(* PLC project ArfBotOS, CODESYS CODESYS V3.5 SP22 Patch 3, author Dale Thomas *)
(* stored: creationDateTime 2026-10-03T14:07:57.8103968, version 1.0.0, modificationDateTime 2026-10-03T14:07:57.6510211, organization Thomas Labs *)
(* https://github.com/dalethomas81/ArfBotOS *)

TYPE ST_CncCmd :
STRUCT
	StartPos: 		SMC_PosInfo;				
	OriConvention: 	SMC_ORI_CONVENTION:=SMC_ORI_CONVENTION.ZYZ;
	Filename: 		STRING:='CNC_FromFile.cnc';
	CoordinateType: DUT_Command_CoordinateType:=DUT_Command_CoordinateType.Variable;
	ArrayIndex: 	INT:=GVL.DEC_START_POS;
	ArrayType: 		DUT_Command_ArrayType:=DUT_Command_ArrayType.StoredPosition;
END_STRUCT
END_TYPE

TYPE DUT_Command :
STRUCT
	CommandType: DUT_CommandType;
	CommandString: STRING(GVL.COMMAND_LEN);
	CommandComment: STRING;
END_STRUCT
END_TYPE

TYPE DUT_Program :
STRUCT
	ProgramName: STRING;
	Commands: ARRAY [GVL.PROG_CMDS_ARR_BEG..GVL.PROG_CMDS_ARR_END] OF DUT_Command;
END_STRUCT
END_TYPE

TYPE DUT_StoredPosition :
STRUCT
	Comment: STRING;
	Position: MC_COORD_REF;
END_STRUCT
END_TYPE

TYPE ST_VisionLocate :
STRUCT
    MaxParts: 		UINT:=1; // max number of parts to locate
    MaxOverlap: 	REAL:=0.0; // max overlap of parts. only needed if MaxParts is greater than zero.
    Score: 			REAL:=0.6; // min score
    ToleranceAngle: REAL:=90.0; // max angle +/- to search
	ResultPosition: UINT:=0; // location to store the results in the vision register array
	TemplateName: 	STRING:='Template.jpg'; // name of the template to search
	ScriptFilename: STRING:='FastTemplateMatching.py'; // name of the script that runs the vision program
END_STRUCT
END_TYPE

TYPE ST_VisionCalibrate :
STRUCT
    CheckerSize: REAL:=25.0; // this value is in user units ex mm
    CheckerXCount: UINT:=6; // count of checker blocks in x coordinate
    CheckerYCount: UINT:=9; // count of checker blocks in y coordinate
END_STRUCT
END_TYPE

TYPE ST_VisionCmd :
STRUCT
    CommandType: DUT_Command_VisionType;
    ImageWidth: UINT:=640; // pixel count in x direction (must be supported by camera)
    ImageHeight: UINT:=400; // pixel coutn in y direction (must be supported by camera)
    Calibrate: ST_VisionCalibrate;
    Locate: ST_VisionLocate;
	Timeout: UDINT:=60; // timeout in seconds
END_STRUCT
END_TYPE

TYPE DUT_VisionRegister EXTENDS DUT_StoredPosition :
STRUCT
	Scaling: REAL;
END_STRUCT
END_TYPE

TYPE DUT_Flags :
STRUCT
	Comment: STRING:='';
	Value: BOOL:=FALSE;
END_STRUCT
END_TYPE

TYPE ST_MoveCmd :
STRUCT
	// common
	MoveType: 					DUT_Command_MoveType:=DUT_Command_MoveType.DirectMove;
	Speed: 						LREAL:=0.0;
	CoordSystem: 				SMC_COORD_SYSTEM:=SMC_COORD_SYSTEM.ACS;
	
	// direct/linear moves
	PositionType: 				DUT_Command_PositionType:=DUT_Command_PositionType.AbsolutePosition;
	CoordinateType: 			DUT_Command_CoordinateType:=DUT_Command_CoordinateType.Literal;
	ArrayIndex: 				UINT:=0;
	ArrayType: 					DUT_Command_ArrayType:=DUT_Command_ArrayType.StoredPosition;
	CoordRef: 					MC_COORD_REF:=(X:=0, Y:=0, Z:=0, A:=0, B:=0, C:=0);
	
	// circular moves
	CircularCoordinateType: 	DUT_Command_CoordinateType:=DUT_Command_CoordinateType.Literal;
	CircularArrayIndex: 		UINT:=0;
	CircularArrayType: 			DUT_Command_ArrayType:=DUT_Command_ArrayType.StoredPosition;
	CircleMode: 				SMC_CIRC_MODE:=SMC_CIRC_MODE.CENTER;
	PathChoice: 				MC_CIRC_PATHCHOICE:=MC_CIRC_PATHCHOICE.CLOCKWISE;
	CoordRef2: 					MC_COORD_REF:=(X:=0, Y:=0, Z:=0, A:=0, B:=0, C:=0);
	
END_STRUCT
END_TYPE

TYPE ST_OutputCmd :
STRUCT
	OutputType: DUT_OutputType;
	OutputTarget: INT;
	OutputValue1: LREAL;
END_STRUCT
END_TYPE

TYPE ST_PauseCmd :
STRUCT
	PauseTime: TIME:=T#1S;
END_STRUCT
END_TYPE

TYPE ST_VarSetCmd :
STRUCT
	ArrayType: DUT_Command_ArrayType;
	ArrayIndex: INT;
	Coordinates: MC_COORD_REF;
	XOperType: DUT_VarSetCmd_OperType;
	YOperType: DUT_VarSetCmd_OperType;
	ZOperType: DUT_VarSetCmd_OperType;
	AOperType: DUT_VarSetCmd_OperType;
	BOperType: DUT_VarSetCmd_OperType;
	COperType: DUT_VarSetCmd_OperType;
END_STRUCT
END_TYPE

TYPE ST_LogicCmdIO :
STRUCT
	Input: ARRAY [GVL.DIG_IN_ARR_BEG..GVL.DIG_IN_ARR_END] OF BOOL;
	Output: ARRAY [GVL.DIG_OUT_ARR_BEG..GVL.DIG_OUT_ARR_END] OF BOOL;
	Pwm: ARRAY [GVL.PWM_OUT_ARR_BEG..GVL.PWM_OUT_ARR_END] OF BYTE;
	Register: ARRAY [GVL.REG_ARR_BEG..GVL.REG_ARR_END] OF UDINT;
	Counter: ARRAY [GVL.REG_ARR_BEG..GVL.REG_ARR_END] OF UDINT;
END_STRUCT
END_TYPE

TYPE ST_LogicCmd :
STRUCT
	IF_Condition : E_LogicIfCondition;
	IF_Condition_Idx: INT;
	IF_Condition_Operator: E_LogicIfConditionOperator;
	IF_Condition_Operator_Value: UDINT;
	THEN_Function: E_LogicFunction;
	THEN_Function_Value: UDINT;
	THEN_Function_Idx: INT;
	ELSE_Function: E_LogicFunction;
	ELSE_Function_Idx: INT;
	ELSE_Function_Value: UDINT;
END_STRUCT
END_TYPE

TYPE ST_Buttons :
STRUCT
	Square: BOOL;
	Triangle: BOOL;
	Circle: BOOL;
	Cross: BOOL;
	Share: BOOL;
	Options: BOOL;
	PS: BOOL;
	Touch: BOOL;
	Mic: BOOL;
END_STRUCT
END_TYPE

TYPE ST_Controller :
STRUCT
	Connected: BOOL;
	Joysticks: ST_Joysticks;
	Buttons: ST_Buttons;
	Dpad: ST_Dpad;
	Triggers: ST_Triggers;
	Trackpads: ST_Trackpads;
	Gyroscope: ST_Gyroscope;
	Accelerometer: ST_Accelerometer;
	Battery: ST_Battery;
END_STRUCT
END_TYPE

TYPE ST_Joystick :
STRUCT
	X: USINT;
	Y: USINT;
	ThreeButton: BOOL;
END_STRUCT
END_TYPE

TYPE ST_Dpad :
STRUCT
	Up: BOOL;
	Down: BOOL;
	Left: BOOL;
	Right: BOOL;
END_STRUCT
END_TYPE

TYPE ST_Trigger :
STRUCT
	One: BOOL;
	Two: USINT;
	TwoButton: BOOL;
END_STRUCT
END_TYPE

TYPE ST_Trackpad :
STRUCT
	ID: USINT;
	Active: BOOL;
	X: UINT;
	Y: UINT;
END_STRUCT
END_TYPE

TYPE ST_Triggers :
STRUCT
	Left: ST_Trigger;
	Right: ST_Trigger;
END_STRUCT
END_TYPE

TYPE ST_Trackpads :
STRUCT
	One: ST_Trackpad;
	Two: ST_Trackpad;
END_STRUCT
END_TYPE

TYPE ST_Joysticks :
STRUCT
	Left: ST_Joystick;
	Right: ST_Joystick;
END_STRUCT
END_TYPE

TYPE ST_Gyroscope :
STRUCT
	Pitch: INT;
	Yaw: INT;
	Roll: INT;
END_STRUCT
END_TYPE

TYPE ST_Accelerometer :
STRUCT
	X: INT;
	Y: INT;
	Z: INT;
END_STRUCT
END_TYPE

TYPE ST_Battery :
STRUCT
	State: USINT;
	Level: USINT;
END_STRUCT
END_TYPE

TYPE DUT_PositionController :
STRUCT
	fKp: LREAL;
	fPartVelPilotControl: LREAL;
	fDeadTime: LREAL;
	fMaxPositionDiff: LREAL;
	fSWMaxVelocity: LREAL;
	fSWMaxAcceleration: LREAL;
	fSWMaxDeceleration: LREAL;
	fSWMaxJerk: LREAL;
END_STRUCT
END_TYPE

TYPE DUT_GroupStatus :
STRUCT
	Valid: BOOL;
	Busy: BOOL;
	Error: BOOL;
	ErrorID: SMC_ERROR;
	GroupMoving: BOOL;
	GroupHoming: BOOL;
	GroupErrorStop: BOOL;
	GroupStandby: BOOL;
	GroupStopping: BOOL;
	GroupDisabled: BOOL;
	TrackingDynamicCS: BOOL;
	InSync: BOOL;
	ActiveMovementId: SMC_Movement_Id;
	FirstReferencedMovementId: SMC_Movement_Id;
	LastAcceptedMovementId: SMC_Movement_Id;
	PositionLag: LREAL;
	OrientationLag: LREAL;
END_STRUCT
END_TYPE

{attribute 'qualified_only'}
{attribute 'strict'}
TYPE E_ControllerPlayerID :
(
	Player1 := 4,
	Player2 := 10,
	Player3 := 21,
	Player4 := 27,
	PlayerAll := 31
);
END_TYPE

{attribute 'qualified_only'}
{attribute 'strict'}
TYPE E_ControllerBrightness :
(
	High := 0,
	Med := 1,
	Low := 2
);
END_TYPE

{attribute 'qualified_only'}
{attribute 'strict'}
TYPE E_ControllerMotor :
(
	Left := 0,
	Right := 1
);
END_TYPE

{attribute 'qualified_only'}
{attribute 'strict'}
TYPE E_ControllerTriggerMode :
(
	Off := 0, // no resistance
	Rigid := 1, // continous resistance
	Pulse := 2, // section resistance
	Rigid_A := 3,
	Rigid_B := 4,
	Rigid_AB := 5,
	Pulse_A := 6,
	Pulse_AB := 7,
	Calibration := 8
);
END_TYPE

{attribute 'qualified_only'}
{attribute 'strict'}
TYPE E_ControllerTrigger :
(
	Left := 0,
	Right := 1
);
END_TYPE

{attribute 'qualified_only'}
{attribute 'strict'}
TYPE E_ControllerTriggerForceParameter :
(
	One := 0,
	Two := 1,
	Three := 2,
	Four := 3,
	Five := 4,
	Six := 5,
	Seven := 6
);
END_TYPE

{attribute 'qualified_only'}
{attribute 'strict'}
TYPE E_Pose :
(
	One := 0,
	Two := 1,
	Three := 2,
	Four := 3,
	Five := 4
);
END_TYPE

TYPE DUT_AxisEnabled :
STRUCT
	J1: BOOL;
	J2: BOOL;
	J3: BOOL;
	J4: BOOL;
	J5: BOOL;
	J6: BOOL;
END_STRUCT
END_TYPE

INTERFACE ITFModule
METHOD M_Start
VAR_INPUT
END_VAR
END_METHOD
METHOD M_Stop
VAR_INPUT
END_VAR
END_METHOD
METHOD M_Home
VAR_INPUT
END_VAR
END_METHOD
METHOD M_Abort
VAR_INPUT
END_VAR
END_METHOD
METHOD M_Hold
VAR_INPUT
END_VAR
END_METHOD
{attribute 'monitoring' := 'variable'}
PROPERTY PropCurrentState : PACK_ML.State
END_PROPERTY
{attribute 'monitoring' := 'variable'}
PROPERTY PropBusy : BOOL
END_PROPERTY
{attribute 'monitoring' := 'variable'}
PROPERTY PropError : BOOL
END_PROPERTY
{attribute 'monitoring' := 'variable'}
PROPERTY PropErrDescription : STRING
END_PROPERTY
END_INTERFACE

TYPE StringByteArray : UNION
  bArray : ARRAY[0..254] OF BYTE;
  sString : STRING(255);
END_UNION;
END_TYPE

PROGRAM _00_Main
VAR
	//
    TaskInfo : POINTER TO CmpIecTask.Task_Info2;
    TaskHandle: CmpIecTask.RTS_IEC_HANDLE;
    Result: CmpIecTask.RTS_IEC_RESULT;
    
	// group handler for all motion fbs
	GroupHandler: FB_GroupHandler;
	
	// tuning
	MoveDistance: LREAL := 5.0;
	MoveRelative: ARRAY[0..5] OF MC_MoveRelative;
	EstimateDeadTime: ARRAY[0..5] OF SMC_EstimateDeadTime;
	TuneStart: ARRAY[0..5] OF BOOL;
	TraceStart: ARRAY[0..5] OF BOOL;
	TraceStop: ARRAY[0..5] OF BOOL;
	SetTuningMoveValues: BOOL:=TRUE;
	fCycleTimeMs: LREAL; (* MainTask / SoftMotion bus cycle, ms *)
	fMeasuredLagMs: ARRAY[0..5] OF LREAL;
	fEstimatedDeadTimeRaw: ARRAY[0..5] OF LREAL; (* unclamped SMC_EstimateDeadTime median *)
	fSuggestedDeadTime: ARRAY[0..5] OF LREAL; (* D in MainTask cycles, clamped to (0, 20] *)
	nDeadTimeSamples: ARRAY[0..5] OF INT;
	bDeadTimeSuggested: ARRAY[0..5] OF BOOL;
	UseSuggestedD: ARRAY[0..5] OF BOOL;
	sDeadTimeHelp: ARRAY[0..5] OF STRING(255);
	fKpPeakLag: ARRAY[0..5] OF LREAL;
	fKpCruiseLag: ARRAY[0..5] OF LREAL;
	fKpFinalLag: ARRAY[0..5] OF LREAL;
	fKpOvershoot: ARRAY[0..5] OF LREAL;
	fKpUndershoot: ARRAY[0..5] OF LREAL;
	nKpReversals: ARRAY[0..5] OF INT;
	nKpVelReversals: ARRAY[0..5] OF INT;
	fSuggestedKp: ARRAY[0..5] OF LREAL;
	bKpSuggested: ARRAY[0..5] OF BOOL;
	UseSuggestedKp: ARRAY[0..5] OF BOOL;
	RaiseKp: ARRAY[0..5] OF BOOL;
	LowerKp: ARRAY[0..5] OF BOOL;
	sKpVerdict: ARRAY[0..5] OF STRING(16);
	sKpHelp: ARRAY[0..5] OF STRING(255);
	
	// homing
	ProcessHome: FB_HomingProcessor;
	HomingStatusText: STRING(255);
	
	// jogging
	ProcessJog: FB_JogProcessor;
	JogStatusText: STRING(255);
	ButtonTextIndex: INT:=0;
	
	// cnc
	VisuStruct3DControl_J: VisuStruct3DControl;
	TrackPosition: FB_PositionTracker;
	
	// program processor
	ProcessPrograms: FB_ProgramProcessor;
	ProcessCommand_ActiveProgram: UINT := 0;
	ActiveCommandDetails: STRING(255):='';
	
	// controller
	Controller: FB_Controller;
	
	//
	EnableRtrig: R_TRIG;
	EnableFtrig: F_TRIG;
	_i, _j, _k: INT;
	BuildTests: BOOL:=FALSE;
	FirstScan: BOOL:=TRUE;

END_VAR

                    
{region "utility"}
    (* Get the current task info *)
    {IF defined (IsSimulationMode)}
        GVL.dwMainInterval := 1000;
    {ELSE}
        TaskHandle := CmpIecTask.IecTaskGetCurrent(ADR(Result));
        TaskInfo := CmpIecTask.IecTaskGetInfo3(TaskHandle, ADR(Result));
        GVL.dwMainInterval := TaskInfo^.dwInterval;
    {END_IF}
    
	GVL.ResetRtrig(CLK:=GVL.Reset);
	IF GVL.ResetRtrig.Q THEN
		GVL.Reset := FALSE;
        AlarmManager.AlarmGlobals.g_AlarmHandler.AcknowledgeAll();
        //AlarmManager.AlarmGlobals.g_AlarmHandler.AcknowledgeAllOfGroup(Alm_AlarmConfiguration_Alarmgroup_IDs.ID_Processors); // only processors
	END_IF
	
	GVL.LicenseStatus();

	IF FirstScan THEN
		M_Init();	
	END_IF
	
	IF BuildTests THEN
		BuildTests := FALSE;
		M_BuildTests();
	END_IF
	
	EnableRtrig(CLK:=GVL.PowerOn);
	EnableFtrig(CLK:=GVL.PowerOn);
	IF EnableRTrig.Q THEN
		GVL.Enable := TRUE;
	END_IF
	IF EnableFTrig.Q THEN
		GVL.Enable := FALSE;
	END_IF
{endregion}
     
{region "methods"}
	_M_GroupHandler();
    _M_Jogging();
    _M_Homing();
    _M_Cnc();
    _M_Processor();
	_M_Controller();
	_M_Tuning();
{endregion}

// do not put anything below this
FirstScan:=FALSE;
                  

METHOD PUBLIC M_Init : BOOL
VAR_INPUT
END_VAR
VAR
    // release
    _hRelease : SysTypes.RTS_IEC_HANDLE;
    _udiReleaseResult : SysTypes.RTS_IEC_RESULT;
    _udiReleaseRead : LWORD;
    _abyRelease : ARRAY[0..80] OF BYTE;
    _iRelease : INT;
    _nRelease : UDINT;
    _pReleaseLen : POINTER TO BYTE;
END_VAR
                          // get release tag to display on HMI
GVL_Version.sRelease := '';
_hRelease := SysFile.SysFileOpen(
    szFile := 'Application/RELEASE',
    am := SysFile.ACCESS_MODE.AM_READ,
    pResult := ADR(_udiReleaseResult));
IF _hRelease <> SysTypes.RTS_INVALID_HANDLE THEN
    _udiReleaseRead := SysFile.SysFileRead(
        hFile := _hRelease,
        pbyBuffer := ADR(_abyRelease),
        ulSize := SIZEOF(_abyRelease) - 1,
        pResult := ADR(_udiReleaseResult));
    SysFile.SysFileClose(_hRelease);

    _nRelease := LWORD_TO_UDINT(_udiReleaseRead);
    IF _nRelease > 80 THEN
        _nRelease := 80;
    END_IF
    WHILE _nRelease > 0 AND
        (_abyRelease[_nRelease - 1] = 10
        OR _abyRelease[_nRelease - 1] = 13
        OR _abyRelease[_nRelease - 1] = 0) DO
        _nRelease := _nRelease - 1;
    END_WHILE

    MemUtils.MemCpy(
        pbyDest := ADR(GVL_Version.sRelease),
        pbySrc := ADR(_abyRelease),
        dwSize := UDINT_TO_DWORD(_nRelease));
    _pReleaseLen := ADR(GVL_Version.sRelease) - 1;
    _pReleaseLen^ := UDINT_TO_BYTE(_nRelease);
    
    GVL_Version.sVersionLine := CONCAT(
        CONCAT('Installer ', GVL_Version.sRelease),
        CONCAT('  PLC ', GVL_Version.sPlcVersion));
    
END_IF
IF GVL_Version.sRelease = '' THEN
    GVL_Version.sVersionLine := 'unknown version';
    
END_IF

// check if arfbot has been initialized
IF NOT PersistentVars.Flags[GVL.INIT_POS_IDX].Value THEN
	// poses
	PersistentVars.Flags[GVL.HOM_TO_POSE_IDX].Value := FALSE;
	PersistentVars.StoredPositions[GVL.POSE_1_IDX].Position.X := 0.0;
	PersistentVars.StoredPositions[GVL.POSE_1_IDX].Position.Y := 0.0;
	PersistentVars.StoredPositions[GVL.POSE_1_IDX].Position.Z := -30.0;
	PersistentVars.StoredPositions[GVL.POSE_1_IDX].Position.A := 0.0;
	PersistentVars.StoredPositions[GVL.POSE_1_IDX].Position.B := -30.0;
	PersistentVars.StoredPositions[GVL.POSE_1_IDX].Position.C := 0.0;
	
	PersistentVars.StoredPositions[GVL.POSE_2_IDX].Position.X := 0.0;
	PersistentVars.StoredPositions[GVL.POSE_2_IDX].Position.Y := 30.0;
	PersistentVars.StoredPositions[GVL.POSE_2_IDX].Position.Z := -30.0;
	PersistentVars.StoredPositions[GVL.POSE_2_IDX].Position.A := 0.0;
	PersistentVars.StoredPositions[GVL.POSE_2_IDX].Position.B := 30.0;
	PersistentVars.StoredPositions[GVL.POSE_2_IDX].Position.C := 0.0;
	
	PersistentVars.StoredPositions[GVL.POSE_3_IDX].Position.X := 0.0;
	PersistentVars.StoredPositions[GVL.POSE_3_IDX].Position.Y := 0.0;
	PersistentVars.StoredPositions[GVL.POSE_3_IDX].Position.Z := 0.0;
	PersistentVars.StoredPositions[GVL.POSE_3_IDX].Position.A := 0.0;
	PersistentVars.StoredPositions[GVL.POSE_3_IDX].Position.B := 90.0;
	PersistentVars.StoredPositions[GVL.POSE_3_IDX].Position.C := 0.0;
	
	PersistentVars.StoredPositions[GVL.POSE_4_IDX].Position.X := 0.0;
	PersistentVars.StoredPositions[GVL.POSE_4_IDX].Position.Y := 0.0;
	PersistentVars.StoredPositions[GVL.POSE_4_IDX].Position.Z := 0.0;
	PersistentVars.StoredPositions[GVL.POSE_4_IDX].Position.A := 0.0;
	PersistentVars.StoredPositions[GVL.POSE_4_IDX].Position.B := 0.0;
	PersistentVars.StoredPositions[GVL.POSE_4_IDX].Position.C := 0.0;
	
	PersistentVars.StoredPositions[GVL.POSE_5_IDX].Position.X := 0.0;
	PersistentVars.StoredPositions[GVL.POSE_5_IDX].Position.Y := 0.0;
	PersistentVars.StoredPositions[GVL.POSE_5_IDX].Position.Z := 0.0;
	PersistentVars.StoredPositions[GVL.POSE_5_IDX].Position.A := 0.0;
	PersistentVars.StoredPositions[GVL.POSE_5_IDX].Position.B := 0.0;
	PersistentVars.StoredPositions[GVL.POSE_5_IDX].Position.C := 0.0;
		 
	// decoder
	PersistentVars.StoredPositions[GVL.DEC_START_POS].Position.X := 300.0; // TODO need to verify all 6 of these
	PersistentVars.StoredPositions[GVL.DEC_START_POS].Position.Y := 0.0;
	PersistentVars.StoredPositions[GVL.DEC_START_POS].Position.Z := -400.0;
	PersistentVars.StoredPositions[GVL.DEC_START_POS].Position.A := 0.0;
	PersistentVars.StoredPositions[GVL.DEC_START_POS].Position.B := 0.0;
	PersistentVars.StoredPositions[GVL.DEC_START_POS].Position.C := 0.0;
	
	// set homing offsets
	PersistentVars.StoredPositions[GVL.HOM_POS_IDX].Position.X := 179.29; // J1 initial home offset
	PersistentVars.StoredPositions[GVL.HOM_POS_IDX].Position.Y := 36.74; // J2 initial home offset
	PersistentVars.StoredPositions[GVL.HOM_POS_IDX].Position.Z := -59.25; // J3 initial home offset
	PersistentVars.StoredPositions[GVL.HOM_POS_IDX].Position.A := -194.38; // J4 initial home offset
	PersistentVars.StoredPositions[GVL.HOM_POS_IDX].Position.B := -102.41; // J5 initial home offset
	PersistentVars.StoredPositions[GVL.HOM_POS_IDX].Position.C := 166.611; // J6 initial home offset
	
	// set speeds
	PersistentVars.StoredPositions[GVL.SPEEDS_IDX].Position.X := 100.0; // max velocity
	PersistentVars.StoredPositions[GVL.SPEEDS_IDX].Position.Y := 1000.0; // max accel/decel
	PersistentVars.StoredPositions[GVL.SPEEDS_IDX].Position.Z := 1000.0; // max jerk
	PersistentVars.StoredPositions[GVL.SPEEDS_IDX].Position.A := 1.0; // velocity factor
	PersistentVars.StoredPositions[GVL.SPEEDS_IDX].Position.B := 0.05; // accel/decel factor
	PersistentVars.StoredPositions[GVL.SPEEDS_IDX].Position.C := 1.0; // jerk factor
	
	//
	M_BuildTests();
		 
	// indicate initialized
	PersistentVars.Flags[GVL.INIT_POS_IDX].Value := TRUE;
END_IF

//
PersistentVars.StoredPositions[GVL.SPEEDS_IDX].Comment := 'vel, acc, jerk, vel fact, acc fact, jerk fact';
PersistentVars.StoredPositions[GVL.HOM_POS_IDX].Comment := 'Home Offsets J1, J2, J3, J4, J5, J6';
PersistentVars.StoredPositions[GVL.DEC_START_POS].Comment := 'NC Decoder Start Position';
PersistentVars.StoredPositions[GVL.TCP_POS_IDX].Comment := 'TCP Offset';
PersistentVars.StoredPositions[GVL.PC2_POS_IDX].Comment := 'PCS 2 Offset';
PersistentVars.StoredPositions[GVL.PC1_POS_IDX].Comment := 'PCS 1 Offset';
PersistentVars.StoredPositions[GVL.MCS_POS_IDX].Comment := 'MCS Offset';

//	 
PersistentVars.StoredPositions[GVL.POSE_1_IDX].Comment := 'Pose 1 coordinates';
PersistentVars.StoredPositions[GVL.POSE_2_IDX].Comment := 'Pose 2 coordinates';
PersistentVars.StoredPositions[GVL.POSE_3_IDX].Comment := 'Pose 3 coordinates';
PersistentVars.StoredPositions[GVL.POSE_4_IDX].Comment := 'Pose 4 coordinates';
PersistentVars.StoredPositions[GVL.POSE_5_IDX].Comment := 'Pose 5 coordinates';

//
PersistentVars.Flags[GVL.HOM_TO_POSE_IDX].Comment := 'Pose 2 After Home';

PersistentVars.Flags[GVL.INIT_DRV_IDX].Comment := 'Drives Initialized';
PersistentVars.Flags[GVL.INIT_DRV_IDX].Value := FALSE;

//
PersistentVars.Flags[GVL.HOME_COMPLETE].Comment := 'Axes Homed';
PersistentVars.Flags[GVL.HOME_COMPLETE].Value := FALSE;

//
PersistentVars.Flags[GVL.INIT_POS_IDX].Comment := 'Variables Intitialized';
                        
END_METHOD

METHOD PRIVATE _M_Homing : BOOL
VAR_INPUT
END_VAR
                          
ProcessHome(
	J1:= IoConfig_Globals.J1, 
	J2:= IoConfig_Globals.J2, 
	J3:= IoConfig_Globals.J3, 
	J4:= IoConfig_Globals.J4, 
	J5:= IoConfig_Globals.J5, 
	J6:= IoConfig_Globals.J6, 
	AxisGroup:= ArfBotAxisGroup,
	GroupHandler:= GroupHandler, 
	Controller:= Controller, 
	J1_Limit:= _10_Robot.rx_j1_limit, 
	J2_Limit:= _10_Robot.rx_j2_limit, 
	J3_Limit:= _10_Robot.rx_j3_limit, 
	J4_Limit:= _10_Robot.rx_j4_limit, 
	J5_Limit:= _10_Robot.rx_j5_limit, 
	J6_Limit:= _10_Robot.rx_j6_limit, 
	Enable:= GVL.Enable, 
	Reset:= GVL.ResetRtrig.Q, 
	StoredPositions:= PersistentVars.StoredPositions,
	VisionRegisters:= PersistentVars.VisionRegisters,
	Flags:= PersistentVars.Flags,
	Done=> , 
	Busy=> , 
	Error=> , 
	ErrorID=> );

IF ProcessHome.Reset THEN
	HomingStatusText := '';
END_IF
IF ProcessHome.Error THEN
	JogStatusText := CONCAT('Homing Processor Error: ',
						CONCAT(TO_STRING(ProcessHome.ErrorID),
						CONCAT(' ', SMC_ErrorString(ProcessHome.ErrorID,
									SMC_Language_Type.english)))) ;
END_IF
                        
END_METHOD

METHOD PRIVATE _M_Processor : BOOL
VAR_INPUT
END_VAR
                          
IF GVL.ResetRtrig.Q THEN
	ProcessPrograms.M_Home();
END_IF

ProcessPrograms(
	Programs:=PersistentVars.Programs,
	StoredPositions:=PersistentVars.StoredPositions,
	VisionRegisters:=PersistentVars.VisionRegisters,
	Flags:=PersistentVars.Flags,
	J1:=IoConfig_Globals.J1, J2:=IoConfig_Globals.J2, J3:=IoConfig_Globals.J3, J4:=IoConfig_Globals.J4, J5:=IoConfig_Globals.J5, J6:=IoConfig_Globals.J6,
	AxisGroup:= ArfBotAxisGroup,
	GroupHandler:= GroupHandler,
	CmdIO:=GVL.CmdIO,
	Enable:= GVL.Enable AND PersistentVars.Flags[GVL.HOME_COMPLETE].Value AND NOT GVL.xActiveAlarm,
	Error=> ,
	StatusText=>);

IF ProcessPrograms.PropBusy THEN
    // for displaying on the HMI
    // PGM: <number> CMD: <number> Type: <type> Command: <command> Comment: <comment>
    ActiveCommandDetails := CONCAT('PGM: ', UINT_TO_STRING(ProcessPrograms.P_CurrentProgram));
    ActiveCommandDetails := CONCAT(ActiveCommandDetails, ' | CMD: ');
    ActiveCommandDetails := CONCAT(ActiveCommandDetails,
                                    // TODO: the "current" index in this case is actually next
                                    // use a SEL here because I dont want to always do "index minus 1" because this would show a -1 on the HMI when Idle and thats gross
                                    UINT_TO_STRING(SEL(ProcessPrograms.P_CurrentCommandIndex <= 0,
                                                        ProcessPrograms.P_CurrentCommandIndex - 1, // FALSE
                                                        0))); // TRUE
    ActiveCommandDetails := CONCAT(ActiveCommandDetails, ' | ');
    ActiveCommandDetails := CONCAT(ActiveCommandDetails, TO_STRING(ProcessPrograms.P_CurrentCommand.CommandType));
    ActiveCommandDetails := CONCAT(ActiveCommandDetails, ': ');
    ActiveCommandDetails := CONCAT(ActiveCommandDetails, ProcessPrograms.P_CurrentCommand.CommandString);
    IF ProcessPrograms.P_CurrentCommand.CommandType = DUT_CommandType.CncCommand THEN
        ActiveCommandDetails := CONCAT(ActiveCommandDetails, ' | G-Code: ');
        ActiveCommandDetails := CONCAT(ActiveCommandDetails, ProcessPrograms.GCodeLines[0]);
    END_IF
    ActiveCommandDetails := CONCAT(ActiveCommandDetails, ' | Comment: ');
    ActiveCommandDetails := CONCAT(ActiveCommandDetails, ProcessPrograms.P_CurrentCommand.CommandComment);
END_IF

// disable all IO when enable drops
IF EnableFtrig.Q THEN
	FOR _i:=GVL.DIG_OUT_ARR_BEG TO GVL.DIG_OUT_ARR_END BY 1 DO
		GVL.CmdIO.Output[_i] := 0;
	END_FOR
	FOR _i:=GVL.PWM_OUT_ARR_BEG TO GVL.PWM_OUT_ARR_END BY 1 DO
		GVL.CmdIO.Pwm[_i] := 0;
	END_FOR
END_IF
                        
END_METHOD

METHOD PRIVATE _M_Cnc : BOOL
VAR_INPUT
END_VAR
VAR
END_VAR
                          // track position of robot end effector to display on hmi
TrackPosition(
	AxisGroup:=ArfBotAxisGroup,
	J1:=IoConfig_Globals.J1,
	J2:=IoConfig_Globals.J2,
	J3:=IoConfig_Globals.J3,
	J4:=IoConfig_Globals.J4,
	J5:=IoConfig_Globals.J5,
	J6:=IoConfig_Globals.J6,
    OriConvention:= GVL.OriConvention,
	VisuStruct3DTrack=>,
	Arm=>,
	Elbow=>,
	Hand=>);
                        
END_METHOD

METHOD PRIVATE _M_Jogging : BOOL
VAR_INPUT
END_VAR
VAR_STAT
	EnableRtrig: R_TRIG;
	CoordSystemLast: SMC_COORD_SYSTEM;
	ABC_AS_ACSLast: BOOL;
END_VAR
                          
// dont get sleepy
ProcessJog(
	AxisGroup:= ArfBotAxisGroup,
	GroupHandler:= GroupHandler,
	Controller:= Controller,
	Enable:= GVL.Enable,
	Reset:= GVL.ResetRtrig.Q,
	StoredPositions:= PersistentVars.StoredPositions,
	VisionRegisters:= PersistentVars.VisionRegisters,
	Flags:= PersistentVars.Flags,
	ABC_as_ACS=>,
	CoordSystem=>, 
	Enabled=>,
	Position=>, 
	Done=> , 
	Busy=> , 
	Error=> , 
	ErrorID=> );
	
// change the button texts on enable or a change of the coordinate system
EnableRtrig(CLK:=ProcessJog.CoordSystem <> CoordSystemLast
				OR ProcessJog.ABC_as_ACS <> ABC_AS_ACSLast);
IF EnableRtrig.Q THEN
	CoordSystemLast := ProcessJog.CoordSystem;
	ABC_AS_ACSLast := ProcessJog.ABC_as_ACS;
	ButtonTextIndex := F_SetJogButtons(ProcessJog.CoordSystem, ProcessJog.ABC_as_ACS);
END_IF
	
//
IF ProcessJog.Reset THEN
	JogStatusText := '';
END_IF
IF ProcessJog.Error THEN
	JogStatusText := CONCAT('Jog Processor Error: ',
						CONCAT(TO_STRING(ProcessJog.ErrorID),
						CONCAT(' ', SMC_ErrorString(ProcessJog.ErrorID,
									SMC_Language_Type.english)))) ;
END_IF
                        
END_METHOD

METHOD PUBLIC M_BuildTests
VAR_INPUT
END_VAR
VAR
	_i, _j, _k: INT;
END_VAR
                          // taught positions referenced by factory programs
PersistentVars.StoredPositions[40].Position.X := -76.81;
PersistentVars.StoredPositions[40].Position.Y := 1.2;
PersistentVars.StoredPositions[40].Position.Z := -24.93;
PersistentVars.StoredPositions[40].Position.A := -4.74;
PersistentVars.StoredPositions[40].Position.B := 62.93;
PersistentVars.StoredPositions[40].Position.C := 24.21;
PersistentVars.StoredPositions[41].Comment := 'Euler Angle Tool Place Position MCS';
PersistentVars.StoredPositions[41].Position.X := 44.39;
PersistentVars.StoredPositions[41].Position.Y := -285.95;
PersistentVars.StoredPositions[41].Position.Z := 310.15;
PersistentVars.StoredPositions[41].Position.A := 96.6;
PersistentVars.StoredPositions[41].Position.B := 177.75;
PersistentVars.StoredPositions[41].Position.C := -174.21;
PersistentVars.StoredPositions[42].Comment := 'Euler Angle Tool Pick Position MCS';
PersistentVars.StoredPositions[42].Position.X := 43.97;
PersistentVars.StoredPositions[42].Position.Y := -280.38;
PersistentVars.StoredPositions[42].Position.Z := 215.24;
PersistentVars.StoredPositions[42].Position.A := 96.61;
PersistentVars.StoredPositions[42].Position.B := 177.75;
PersistentVars.StoredPositions[42].Position.C := -174.22;

//
FOR _i := GVL.PROG_CMDS_ARR_BEG TO GVL.PROG_CMDS_ARR_END BY 1 DO
	PersistentVars.Programs[0].Commands[_i].CommandType := DUT_CommandType.Disabled;
	PersistentVars.Programs[0].Commands[_i].CommandString := '';
	PersistentVars.Programs[0].Commands[_i].CommandComment := '';
END_FOR
PersistentVars.Programs[0].ProgramName := 'Pick and Place Euler Angle Tool';
PersistentVars.Programs[0].Commands[0].CommandType := DUT_CommandType.MoveCommand;
PersistentVars.Programs[0].Commands[0].CommandString := 'DIR ABS 50.0 ACS VAR STO 35 ';
PersistentVars.Programs[0].Commands[0].CommandComment := 'take on a pose';
PersistentVars.Programs[0].Commands[1].CommandType := DUT_CommandType.VarSetCommand;
PersistentVars.Programs[0].Commands[1].CommandString := 'STO 46 E 0.0 E 0.0 E 0.0 E 0.0 E 0.0 E 0.0 ';
PersistentVars.Programs[0].Commands[1].CommandComment := 'Rotate TCP according to ZYZ convention';
PersistentVars.Programs[0].Commands[3].CommandType := DUT_CommandType.LogicCommand;
PersistentVars.Programs[0].Commands[3].CommandString := 'IF REGISTER 40 EQU 0 THEN JUMP 5 ELSE JUMP 12 ';
PersistentVars.Programs[0].Commands[3].CommandComment := 'determine if pick or place';
PersistentVars.Programs[0].Commands[5].CommandType := DUT_CommandType.MoveCommand;
PersistentVars.Programs[0].Commands[5].CommandString := 'DIR ABS 50.0 MCS VAR STO 42 ';
PersistentVars.Programs[0].Commands[5].CommandComment := 'go to euler angle tool down position';
PersistentVars.Programs[0].Commands[6].CommandType := DUT_CommandType.OutputCommand;
PersistentVars.Programs[0].Commands[6].CommandString := 'DIG 0 1.0 ';
PersistentVars.Programs[0].Commands[6].CommandComment := 'open gripper';
PersistentVars.Programs[0].Commands[7].CommandType := DUT_CommandType.MoveCommand;
PersistentVars.Programs[0].Commands[7].CommandString := 'LIN REL 20.0 TCS LIT 0.0 0.0 25.0 0.0 0.0 0.0 ';
PersistentVars.Programs[0].Commands[7].CommandComment := 'move onto euler angle tool';
PersistentVars.Programs[0].Commands[8].CommandType := DUT_CommandType.OutputCommand;
PersistentVars.Programs[0].Commands[8].CommandString := 'DIG 0 0.0 ';
PersistentVars.Programs[0].Commands[8].CommandComment := 'close gripper';
PersistentVars.Programs[0].Commands[9].CommandType := DUT_CommandType.MoveCommand;
PersistentVars.Programs[0].Commands[9].CommandString := 'LIN REL 20.0 TCS LIT 0.0 0.0 -120.0 0.0 0.0 0.0 ';
PersistentVars.Programs[0].Commands[9].CommandComment := 'pull out tool';
PersistentVars.Programs[0].Commands[10].CommandType := DUT_CommandType.LogicCommand;
PersistentVars.Programs[0].Commands[10].CommandString := 'IF PASS THEN JUMP 16 ';
PersistentVars.Programs[0].Commands[12].CommandType := DUT_CommandType.MoveCommand;
PersistentVars.Programs[0].Commands[12].CommandString := 'DIR ABS 50.0 MCS VAR STO 41 ';
PersistentVars.Programs[0].Commands[12].CommandComment := 'go to euler angle tool up position';
PersistentVars.Programs[0].Commands[13].CommandType := DUT_CommandType.MoveCommand;
PersistentVars.Programs[0].Commands[13].CommandString := 'LIN REL 20.0 TCS LIT 0.0 0.0 120.0 0.0 0.0 0.0 ';
PersistentVars.Programs[0].Commands[13].CommandComment := 'push tool in';
PersistentVars.Programs[0].Commands[14].CommandType := DUT_CommandType.OutputCommand;
PersistentVars.Programs[0].Commands[14].CommandString := 'DIG 0 1.0 ';
PersistentVars.Programs[0].Commands[14].CommandComment := 'open gripper';
PersistentVars.Programs[0].Commands[15].CommandType := DUT_CommandType.MoveCommand;
PersistentVars.Programs[0].Commands[15].CommandString := 'LIN REL 20.0 TCS LIT 0.0 0.0 -25.0 0.0 0.0 0.0 ';
PersistentVars.Programs[0].Commands[15].CommandComment := 'move away from euler angle tool';

//
FOR _i := GVL.PROG_CMDS_ARR_BEG TO GVL.PROG_CMDS_ARR_END BY 1 DO
	PersistentVars.Programs[1].Commands[_i].CommandType := DUT_CommandType.Disabled;
	PersistentVars.Programs[1].Commands[_i].CommandString := '';
	PersistentVars.Programs[1].Commands[_i].CommandComment := '';
END_FOR
PersistentVars.Programs[1].ProgramName := 'Vision Pick and Place';
PersistentVars.Programs[1].Commands[0].CommandType := DUT_CommandType.VarSetCommand;
PersistentVars.Programs[1].Commands[0].CommandString := 'STO 46 E 0.0 E 0.0 E 0.0 E 0.0 E 0.0 E 90.0 ';
PersistentVars.Programs[1].Commands[0].CommandComment := 'Rotate TCP according to ZYZ convention';
PersistentVars.Programs[1].Commands[1].CommandType := DUT_CommandType.MoveCommand;
PersistentVars.Programs[1].Commands[1].CommandString := 'DIR ABS 60.0 ACS VAR STO 40 ';
PersistentVars.Programs[1].Commands[1].CommandComment := 'Take a pose';
PersistentVars.Programs[1].Commands[2].CommandType := DUT_CommandType.VisionCommand;
PersistentVars.Programs[1].Commands[2].CommandString := 'LOC 640 400 15 1 0.0 0.6 180.0 0 Pen.jpg FastTemplateMatching.py ';
PersistentVars.Programs[1].Commands[2].CommandComment := 'Find the object and store the result';
PersistentVars.Programs[1].Commands[3].CommandType := DUT_CommandType.VarSetCommand;
PersistentVars.Programs[1].Commands[3].CommandString := 'VIS 0 M -1.0 M -1.0 E -20.0 M -1.0 N 0.0 N 0.0 ';
PersistentVars.Programs[1].Commands[3].CommandComment := 'Rotate x and y to line up with TCP';
PersistentVars.Programs[1].Commands[4].CommandType := DUT_CommandType.MoveCommand;
PersistentVars.Programs[1].Commands[4].CommandString := 'DIR ABS 50.0 PC1 VAR VIS 0 ';
PersistentVars.Programs[1].Commands[4].CommandComment := 'Move over the object';
PersistentVars.Programs[1].Commands[5].CommandType := DUT_CommandType.OutputCommand;
PersistentVars.Programs[1].Commands[5].CommandString := 'DIG 0 1.0 ';
PersistentVars.Programs[1].Commands[5].CommandComment := 'Open the Gripper';
PersistentVars.Programs[1].Commands[6].CommandType := DUT_CommandType.MoveCommand;
PersistentVars.Programs[1].Commands[6].CommandString := 'LIN REL 50.0 TCS LIT 0.0 0.0 20.0 0.0 0.0 0.0 ';
PersistentVars.Programs[1].Commands[6].CommandComment := 'Move down to the object';
PersistentVars.Programs[1].Commands[7].CommandType := DUT_CommandType.OutputCommand;
PersistentVars.Programs[1].Commands[7].CommandString := 'DIG 0 0.0 ';
PersistentVars.Programs[1].Commands[7].CommandComment := 'Close the Gripper';
PersistentVars.Programs[1].Commands[8].CommandType := DUT_CommandType.PauseCommand;
PersistentVars.Programs[1].Commands[8].CommandString := 'T#1s';
PersistentVars.Programs[1].Commands[8].CommandComment := 'Pause while the gripper closes';
PersistentVars.Programs[1].Commands[9].CommandType := DUT_CommandType.MoveCommand;
PersistentVars.Programs[1].Commands[9].CommandString := 'LIN REL 50.0 TCS LIT 0.0 0.0 -20.0 0.0 0.0 0.0 ';
PersistentVars.Programs[1].Commands[9].CommandComment := 'Pick up the object';
PersistentVars.Programs[1].Commands[10].CommandType := DUT_CommandType.MoveCommand;
PersistentVars.Programs[1].Commands[10].CommandString := 'DIR ABS 50.0 PC1 LIT 0.0 0.0 -50.0 0.0 0.0 90.0 ';
PersistentVars.Programs[1].Commands[10].CommandComment := 'Move to drop position';
PersistentVars.Programs[1].Commands[11].CommandType := DUT_CommandType.OutputCommand;
PersistentVars.Programs[1].Commands[11].CommandString := 'DIG 0 1.0 ';
PersistentVars.Programs[1].Commands[11].CommandComment := 'Open the Gripper';

//
FOR _i := GVL.PROG_CMDS_ARR_BEG TO GVL.PROG_CMDS_ARR_END BY 1 DO
	PersistentVars.Programs[2].Commands[_i].CommandType := DUT_CommandType.Disabled;
	PersistentVars.Programs[2].Commands[_i].CommandString := '';
	PersistentVars.Programs[2].Commands[_i].CommandComment := '';
END_FOR
PersistentVars.Programs[2].ProgramName := 'PCS1 Corners';
PersistentVars.Programs[2].Commands[0].CommandType := DUT_CommandType.VarSetCommand;
PersistentVars.Programs[2].Commands[0].CommandString := 'STO 46 E 0.0 E 0.0 E 0.0 E 180.0 E 180.0 E 0.0 ';
PersistentVars.Programs[2].Commands[0].CommandComment := 'Rotate TCP according to ZYZ convention';
PersistentVars.Programs[2].Commands[1].CommandType := DUT_CommandType.VarSetCommand;
PersistentVars.Programs[2].Commands[1].CommandString := 'STO 48 E 282.23 E -0066.77 E 0195.00 E 0.0 E 0.0 E -0030.00 ';
PersistentVars.Programs[2].Commands[2].CommandType := DUT_CommandType.MoveCommand;
PersistentVars.Programs[2].Commands[2].CommandString := 'DIR ABS 050 PC1 LIT 0 0 0 0 0 0';
PersistentVars.Programs[2].Commands[3].CommandType := DUT_CommandType.MoveCommand;
PersistentVars.Programs[2].Commands[3].CommandString := 'LIN REL 100 TCS LIT 0.0 200.0 0.0 0.0 0.0 0.0';
PersistentVars.Programs[2].Commands[4].CommandType := DUT_CommandType.MoveCommand;
PersistentVars.Programs[2].Commands[4].CommandString := 'LIN REL 100 TCS LIT 00125.00 00000.00 00000.00 00000.00 00000.00 00000.00';
PersistentVars.Programs[2].Commands[5].CommandType := DUT_CommandType.MoveCommand;
PersistentVars.Programs[2].Commands[5].CommandString := 'LIN REL 100 TCS LIT 00000.00 -0200.00 00000.00 00000.00 00000.00 00000.00';
PersistentVars.Programs[2].Commands[6].CommandType := DUT_CommandType.MoveCommand;
PersistentVars.Programs[2].Commands[6].CommandString := 'LIN REL 100 TCS LIT -0125.00 00000.00 00000.00 00000.00 00000.00 00000.00';
PersistentVars.Programs[2].Commands[7].CommandType := DUT_CommandType.MoveCommand;
PersistentVars.Programs[2].Commands[7].CommandString := 'DIR ABS 050 ACS LIT +00 +30 -30 +00 +30 +00';

//
FOR _i := GVL.PROG_CMDS_ARR_BEG TO GVL.PROG_CMDS_ARR_END BY 1 DO
	PersistentVars.Programs[3].Commands[_i].CommandType := DUT_CommandType.Disabled;
	PersistentVars.Programs[3].Commands[_i].CommandString := '';
	PersistentVars.Programs[3].Commands[_i].CommandComment := '';
END_FOR
PersistentVars.Programs[3].ProgramName := 'Cnc Validation';
PersistentVars.Programs[3].Commands[0].CommandType := DUT_CommandType.MoveCommand;
PersistentVars.Programs[3].Commands[0].CommandString := 'DIR ABS 30.0 ACS VAR STO 34 ';
PersistentVars.Programs[3].Commands[1].CommandType := DUT_CommandType.CncCommand;
PersistentVars.Programs[3].Commands[1].CommandString := 'CNC_FromFile.cnc';

//
FOR _i := GVL.PROG_CMDS_ARR_BEG TO GVL.PROG_CMDS_ARR_END BY 1 DO
	PersistentVars.Programs[4].Commands[_i].CommandType := DUT_CommandType.Disabled;
	PersistentVars.Programs[4].Commands[_i].CommandString := '';
	PersistentVars.Programs[4].Commands[_i].CommandComment := '';
END_FOR
PersistentVars.Programs[4].ProgramName := 'Vision Validation';
PersistentVars.Programs[4].Commands[0].CommandType := DUT_CommandType.VisionCommand;
PersistentVars.Programs[4].Commands[0].CommandString := 'LOC 640 400 60 1 0.0 0.8 30.0 10 Template.jpg FastTemplateMatching.py';
PersistentVars.Programs[4].Commands[1].CommandType := DUT_CommandType.VisionCommand;
PersistentVars.Programs[4].Commands[1].CommandString := 'LOC 640 400 60 1 0.0 0.8 30.0 4 strippers2.jpg FastTemplateMatching.py';

//
FOR _i := GVL.PROG_CMDS_ARR_BEG TO GVL.PROG_CMDS_ARR_END BY 1 DO
	PersistentVars.Programs[5].Commands[_i].CommandType := DUT_CommandType.Disabled;
	PersistentVars.Programs[5].Commands[_i].CommandString := '';
	PersistentVars.Programs[5].Commands[_i].CommandComment := '';
END_FOR
PersistentVars.Programs[5].ProgramName := 'VarSet Validation';
PersistentVars.Programs[5].Commands[0].CommandType := DUT_CommandType.VarSetCommand;
PersistentVars.Programs[5].Commands[0].CommandString := 'STO 1 E 6.0 E 5.0 E 4.0 E 3.0 E 2.0 E 1.0 ';
PersistentVars.Programs[5].Commands[1].CommandType := DUT_CommandType.VarSetCommand;
PersistentVars.Programs[5].Commands[1].CommandString := 'VIS 2 1 2 3 4 5 6';
PersistentVars.Programs[5].Commands[2].CommandType := DUT_CommandType.VarSetCommand;
PersistentVars.Programs[5].Commands[2].CommandString := 'FLG 3 1';

//
FOR _i := GVL.PROG_CMDS_ARR_BEG TO GVL.PROG_CMDS_ARR_END BY 1 DO
	PersistentVars.Programs[6].Commands[_i].CommandType := DUT_CommandType.Disabled;
	PersistentVars.Programs[6].Commands[_i].CommandString := '';
	PersistentVars.Programs[6].Commands[_i].CommandComment := '';
END_FOR
PersistentVars.Programs[6].ProgramName := 'Logic Validation';
PersistentVars.Programs[6].Commands[0].CommandType := DUT_CommandType.LogicCommand;
PersistentVars.Programs[6].Commands[0].CommandString := 'IF INPUT 1 EQU 1 THEN OUTPUT 1 1 ELSE OUTPUT 1 0';
PersistentVars.Programs[6].Commands[1].CommandType := DUT_CommandType.LogicCommand;
PersistentVars.Programs[6].Commands[1].CommandString := 'IF INPUT 1 EQU 1 THEN CNTUP 1 ELSE CNTUP 2';
PersistentVars.Programs[6].Commands[2].CommandType := DUT_CommandType.LogicCommand;
PersistentVars.Programs[6].Commands[2].CommandString := 'IF COUNTER 2 GRE 10 THEN NOP ELSE JUMP 0';

//
FOR _i := GVL.PROG_CMDS_ARR_BEG TO GVL.PROG_CMDS_ARR_END BY 1 DO
	PersistentVars.Programs[7].Commands[_i].CommandType := DUT_CommandType.Disabled;
	PersistentVars.Programs[7].Commands[_i].CommandString := '';
	PersistentVars.Programs[7].Commands[_i].CommandComment := '';
END_FOR
PersistentVars.Programs[7].ProgramName := 'Euler Angles Demo';
PersistentVars.Programs[7].Commands[0].CommandType := DUT_CommandType.LogicCommand;
PersistentVars.Programs[7].Commands[0].CommandString := 'IF PASS THEN REGISTER 40 0 ';
PersistentVars.Programs[7].Commands[0].CommandComment := 'Set pick/place register to pick tool';
PersistentVars.Programs[7].Commands[1].CommandType := DUT_CommandType.LogicCommand;
PersistentVars.Programs[7].Commands[1].CommandString := 'IF PASS THEN CALL 0 ';
PersistentVars.Programs[7].Commands[1].CommandComment := 'Call pick and place program';
PersistentVars.Programs[7].Commands[3].CommandType := DUT_CommandType.LogicCommand;
PersistentVars.Programs[7].Commands[3].CommandString := 'IF COUNTER 7 EQU 0 THEN NOP ELSE JUMP 7 ';
PersistentVars.Programs[7].Commands[3].CommandComment := 'apply or jump over';
PersistentVars.Programs[7].Commands[4].CommandType := DUT_CommandType.VarSetCommand;
PersistentVars.Programs[7].Commands[4].CommandString := 'STO 46 E 0.0 E 0.0 E 70.0 E 0.0 E 0.0 E 0.0 ';
PersistentVars.Programs[7].Commands[4].CommandComment := 'offset TCP Z';
PersistentVars.Programs[7].Commands[5].CommandType := DUT_CommandType.LogicCommand;
PersistentVars.Programs[7].Commands[5].CommandString := 'IF PASS THEN JUMP 19 ';
PersistentVars.Programs[7].Commands[5].CommandComment := 'go to move commands';
PersistentVars.Programs[7].Commands[7].CommandType := DUT_CommandType.LogicCommand;
PersistentVars.Programs[7].Commands[7].CommandString := 'IF COUNTER 7 EQU 1 THEN NOP ELSE JUMP 11 ';
PersistentVars.Programs[7].Commands[7].CommandComment := 'apply or jump over';
PersistentVars.Programs[7].Commands[8].CommandType := DUT_CommandType.VarSetCommand;
PersistentVars.Programs[7].Commands[8].CommandString := 'STO 46 E 0.0 E 0.0 E 170.0 E 0.0 E 0.0 E 0.0 ';
PersistentVars.Programs[7].Commands[8].CommandComment := 'offset TCP Z';
PersistentVars.Programs[7].Commands[9].CommandType := DUT_CommandType.LogicCommand;
PersistentVars.Programs[7].Commands[9].CommandString := 'IF PASS THEN JUMP 19 ';
PersistentVars.Programs[7].Commands[9].CommandComment := 'go to move commands';
PersistentVars.Programs[7].Commands[11].CommandType := DUT_CommandType.LogicCommand;
PersistentVars.Programs[7].Commands[11].CommandString := 'IF COUNTER 7 EQU 2 THEN NOP ELSE JUMP 15 ';
PersistentVars.Programs[7].Commands[11].CommandComment := 'apply or jump over';
PersistentVars.Programs[7].Commands[12].CommandType := DUT_CommandType.VarSetCommand;
PersistentVars.Programs[7].Commands[12].CommandString := 'STO 46 E 0.0 E -100.0 E 70.0 E 0.0 E 0.0 E 0.0 ';
PersistentVars.Programs[7].Commands[12].CommandComment := 'offset TCP X and Y';
PersistentVars.Programs[7].Commands[13].CommandType := DUT_CommandType.LogicCommand;
PersistentVars.Programs[7].Commands[13].CommandString := 'IF PASS THEN JUMP 19 ';
PersistentVars.Programs[7].Commands[13].CommandComment := 'go to move commands';
PersistentVars.Programs[7].Commands[15].CommandType := DUT_CommandType.LogicCommand;
PersistentVars.Programs[7].Commands[15].CommandString := 'IF COUNTER 7 EQU 3 THEN NOP ELSE JUMP 29 ';
PersistentVars.Programs[7].Commands[15].CommandComment := 'apply or jump over';
PersistentVars.Programs[7].Commands[16].CommandType := DUT_CommandType.VarSetCommand;
PersistentVars.Programs[7].Commands[16].CommandString := 'STO 46 E 100.0 E 0.0 E 70.0 E 0.0 E 0.0 E 0.0 ';
PersistentVars.Programs[7].Commands[16].CommandComment := 'offset TCP X and Z';
PersistentVars.Programs[7].Commands[17].CommandType := DUT_CommandType.LogicCommand;
PersistentVars.Programs[7].Commands[17].CommandString := 'IF PASS THEN JUMP 19 ';
PersistentVars.Programs[7].Commands[17].CommandComment := 'go to move commands';
PersistentVars.Programs[7].Commands[19].CommandType := DUT_CommandType.MoveCommand;
PersistentVars.Programs[7].Commands[19].CommandString := 'DIR ABS 50.0 ACS VAR STO 35 ';
PersistentVars.Programs[7].Commands[19].CommandComment := 'take on a pose';
PersistentVars.Programs[7].Commands[20].CommandType := DUT_CommandType.MoveCommand;
PersistentVars.Programs[7].Commands[20].CommandString := 'LIN ABS 70.0 TCS LIT 0.0 0.0 0.0 0.0 0.0 -45.0 ';
PersistentVars.Programs[7].Commands[20].CommandComment := 'rotate TCP Z with ZYZ convention';
PersistentVars.Programs[7].Commands[21].CommandType := DUT_CommandType.MoveCommand;
PersistentVars.Programs[7].Commands[21].CommandString := 'LIN ABS 70.0 TCS LIT 0.0 0.0 0.0 0.0 -30.0 0.0 ';
PersistentVars.Programs[7].Commands[21].CommandComment := 'rotate around TCP Y with ZYZ convention';
PersistentVars.Programs[7].Commands[22].CommandType := DUT_CommandType.MoveCommand;
PersistentVars.Programs[7].Commands[22].CommandString := 'LIN ABS 70.0 TCS LIT 0.0 0.0 0.0 90.0 30.0 -90.0 ';
PersistentVars.Programs[7].Commands[22].CommandComment := 'rotate around TCP X with ZYZ convention';
PersistentVars.Programs[7].Commands[23].CommandType := DUT_CommandType.MoveCommand;
PersistentVars.Programs[7].Commands[23].CommandString := 'LIN ABS 70.0 TCS LIT 0.0 0.0 0.0 90.0 -30.0 -90.0 ';
PersistentVars.Programs[7].Commands[23].CommandComment := 'rotate around TCP X with ZYZ convention';
PersistentVars.Programs[7].Commands[24].CommandType := DUT_CommandType.MoveCommand;
PersistentVars.Programs[7].Commands[24].CommandString := 'LIN ABS 70.0 TCS LIT 0.0 0.0 0.0 0.0 30.0 0.0 ';
PersistentVars.Programs[7].Commands[24].CommandComment := 'rotate around TCP Y with ZYZ convention';
PersistentVars.Programs[7].Commands[25].CommandType := DUT_CommandType.MoveCommand;
PersistentVars.Programs[7].Commands[25].CommandString := 'DIR ABS 70.0 ACS VAR STO 35 ';
PersistentVars.Programs[7].Commands[25].CommandComment := 'take on a pose';
PersistentVars.Programs[7].Commands[27].CommandType := DUT_CommandType.LogicCommand;
PersistentVars.Programs[7].Commands[27].CommandString := 'IF PASS THEN CNTUP 7 ';
PersistentVars.Programs[7].Commands[27].CommandComment := 'count up counter';
PersistentVars.Programs[7].Commands[28].CommandType := DUT_CommandType.LogicCommand;
PersistentVars.Programs[7].Commands[28].CommandString := 'IF PASS THEN JUMP 3 ';
PersistentVars.Programs[7].Commands[28].CommandComment := 'go back to start';
PersistentVars.Programs[7].Commands[29].CommandType := DUT_CommandType.LogicCommand;
PersistentVars.Programs[7].Commands[29].CommandString := 'IF PASS THEN CNTRST 7 ';
PersistentVars.Programs[7].Commands[29].CommandComment := 'reset counter back to 0';
PersistentVars.Programs[7].Commands[31].CommandType := DUT_CommandType.LogicCommand;
PersistentVars.Programs[7].Commands[31].CommandString := 'IF PASS THEN REGISTER 40 1 ';
PersistentVars.Programs[7].Commands[31].CommandComment := 'Set pick/place register to place tool';
PersistentVars.Programs[7].Commands[32].CommandType := DUT_CommandType.LogicCommand;
PersistentVars.Programs[7].Commands[32].CommandString := 'IF PASS THEN CALL 0 ';
PersistentVars.Programs[7].Commands[32].CommandComment := 'Call pick and place program';

//
FOR _i := GVL.PROG_CMDS_ARR_BEG TO GVL.PROG_CMDS_ARR_END BY 1 DO
	PersistentVars.Programs[10].Commands[_i].CommandType := DUT_CommandType.Disabled;
	PersistentVars.Programs[10].Commands[_i].CommandString := '';
	PersistentVars.Programs[10].Commands[_i].CommandComment := '';
END_FOR
PersistentVars.Programs[10].ProgramName := 'Pick Glow Stick';
PersistentVars.Programs[10].Commands[0].CommandType := DUT_CommandType.LogicCommand;
PersistentVars.Programs[10].Commands[0].CommandString := 'IF REGISTER 2 EQU 0 THEN NOP ELSE JUMP 5 ';
PersistentVars.Programs[10].Commands[0].CommandComment := 'check if initialized';
PersistentVars.Programs[10].Commands[1].CommandType := DUT_CommandType.VarSetCommand;
PersistentVars.Programs[10].Commands[1].CommandString := 'STO 0 E 0.0 E 0.0 E 0.0 E 0.0 E 0.0 E 0.0 ';
PersistentVars.Programs[10].Commands[1].CommandComment := 'clear out the tcp position';
PersistentVars.Programs[10].Commands[2].CommandType := DUT_CommandType.LogicCommand;
PersistentVars.Programs[10].Commands[2].CommandString := 'IF PASS THEN CNTRST 0 ';
PersistentVars.Programs[10].Commands[2].CommandComment := 'clear column counter';
PersistentVars.Programs[10].Commands[3].CommandType := DUT_CommandType.LogicCommand;
PersistentVars.Programs[10].Commands[3].CommandString := 'IF PASS THEN CNTRST 1 ';
PersistentVars.Programs[10].Commands[3].CommandComment := 'clear row counter';
PersistentVars.Programs[10].Commands[4].CommandType := DUT_CommandType.LogicCommand;
PersistentVars.Programs[10].Commands[4].CommandString := 'IF PASS THEN REGISTER 2 1 ';
PersistentVars.Programs[10].Commands[4].CommandComment := 'mark data initialized';
PersistentVars.Programs[10].Commands[6].CommandType := DUT_CommandType.MoveCommand;
PersistentVars.Programs[10].Commands[6].CommandString := 'DIR ABS 50.0 ACS VAR STO 34 ';
PersistentVars.Programs[10].Commands[6].CommandComment := 'take on a pose';
PersistentVars.Programs[10].Commands[7].CommandType := DUT_CommandType.OutputCommand;
PersistentVars.Programs[10].Commands[7].CommandString := 'DIG 0 1.0 ';
PersistentVars.Programs[10].Commands[7].CommandComment := 'open gripper';
PersistentVars.Programs[10].Commands[8].CommandType := DUT_CommandType.MoveCommand;
PersistentVars.Programs[10].Commands[8].CommandString := 'LIN ABS 50.0 PC1 VAR STO 0 ';
PersistentVars.Programs[10].Commands[8].CommandComment := 'go to the pick position in PCS1';
PersistentVars.Programs[10].Commands[9].CommandType := DUT_CommandType.MoveCommand;
PersistentVars.Programs[10].Commands[9].CommandString := 'LIN REL 50.0 TCS LIT 0.0 0.0 10.0 0.0 0.0 0.0 ';
PersistentVars.Programs[10].Commands[9].CommandComment := 'move into glow stick';
PersistentVars.Programs[10].Commands[10].CommandType := DUT_CommandType.OutputCommand;
PersistentVars.Programs[10].Commands[10].CommandString := 'DIG 0 0.0 ';
PersistentVars.Programs[10].Commands[10].CommandComment := 'close gripper';
PersistentVars.Programs[10].Commands[11].CommandType := DUT_CommandType.MoveCommand;
PersistentVars.Programs[10].Commands[11].CommandString := 'LIN REL 50.0 TCS LIT 160.0 0.0 0.0 0.0 0.0 0.0 ';
PersistentVars.Programs[10].Commands[11].CommandComment := 'pick glow stick out of nest';
PersistentVars.Programs[10].Commands[12].CommandType := DUT_CommandType.MoveCommand;
PersistentVars.Programs[10].Commands[12].CommandString := 'LIN ABS 50.0 PC2 LIT 0.0 0.0 0.0 0.0 0.0 0.0 ';
PersistentVars.Programs[10].Commands[12].CommandComment := 'go to the home position of PCS2';
PersistentVars.Programs[10].Commands[13].CommandType := DUT_CommandType.MoveCommand;
PersistentVars.Programs[10].Commands[13].CommandString := 'LIN REL 50.0 TCS LIT 0.0 0.0 50.0 0.0 0.0 0.0 ';
PersistentVars.Programs[10].Commands[13].CommandComment := 'move into drop position';
PersistentVars.Programs[10].Commands[14].CommandType := DUT_CommandType.OutputCommand;
PersistentVars.Programs[10].Commands[14].CommandString := 'DIG 0 1.0 ';
PersistentVars.Programs[10].Commands[14].CommandComment := 'open gripper';
PersistentVars.Programs[10].Commands[15].CommandType := DUT_CommandType.MoveCommand;
PersistentVars.Programs[10].Commands[15].CommandString := 'LIN ABS 50.0 PC2 LIT 0.0 0.0 0.0 0.0 0.0 0.0 ';
PersistentVars.Programs[10].Commands[15].CommandComment := 'go to the home position of PCS2';
PersistentVars.Programs[10].Commands[17].CommandType := DUT_CommandType.LogicCommand;
PersistentVars.Programs[10].Commands[17].CommandString := 'IF COUNTER 0 LES 3 THEN CNTUP 0 ELSE JUMP 21 ';
PersistentVars.Programs[10].Commands[17].CommandComment := 'increment the column counter';
PersistentVars.Programs[10].Commands[18].CommandType := DUT_CommandType.VarSetCommand;
PersistentVars.Programs[10].Commands[18].CommandString := 'STO 0 N 0.0 A 20.0 N 0.0 N 0.0 N 0.0 N 0.0 ';
PersistentVars.Programs[10].Commands[18].CommandComment := 'add the column width';
PersistentVars.Programs[10].Commands[20].CommandType := DUT_CommandType.LogicCommand;
PersistentVars.Programs[10].Commands[20].CommandString := 'IF PASS THEN JUMP 24 ';
PersistentVars.Programs[10].Commands[20].CommandComment := 'jump over the counter operations';
PersistentVars.Programs[10].Commands[21].CommandType := DUT_CommandType.LogicCommand;
PersistentVars.Programs[10].Commands[21].CommandString := 'IF PASS THEN CNTRST 0 ';
PersistentVars.Programs[10].Commands[21].CommandComment := 'reset the column counter';
PersistentVars.Programs[10].Commands[22].CommandType := DUT_CommandType.LogicCommand;
PersistentVars.Programs[10].Commands[22].CommandString := 'IF PASS THEN CNTUP 1 ';
PersistentVars.Programs[10].Commands[22].CommandComment := 'increment the row counter';
PersistentVars.Programs[10].Commands[23].CommandType := DUT_CommandType.VarSetCommand;
PersistentVars.Programs[10].Commands[23].CommandString := 'STO 0 N 0.0 E 0.0 A 15.0 N 0.0 N 0.0 N 0.0 ';
PersistentVars.Programs[10].Commands[23].CommandComment := 'add the row width. clear column.';

//
FOR _i := GVL.PROG_CMDS_ARR_BEG TO GVL.PROG_CMDS_ARR_END BY 1 DO
	PersistentVars.Programs[15].Commands[_i].CommandType := DUT_CommandType.Disabled;
	PersistentVars.Programs[15].Commands[_i].CommandString := '';
	PersistentVars.Programs[15].Commands[_i].CommandComment := '';
END_FOR
PersistentVars.Programs[15].ProgramName := 'Gimbal 1';
PersistentVars.Programs[15].Commands[0].CommandType := DUT_CommandType.VarSetCommand;
PersistentVars.Programs[15].Commands[0].CommandString := 'STO 43 N 0.0 E 250.0 E 250.0 N 0.0 E 1.0e-2 E 1.0e-1 ';
PersistentVars.Programs[15].Commands[0].CommandComment := 'set velocity, acceleration, and jerk';
PersistentVars.Programs[15].Commands[1].CommandType := DUT_CommandType.VarSetCommand;
PersistentVars.Programs[15].Commands[1].CommandString := 'STO 43 E 100.0 E 1000.0 E 1000.0 E 1.0 E 1.0 E 1.0 ';
PersistentVars.Programs[15].Commands[1].CommandComment := 'set velocity, acceleration, and jerk';
PersistentVars.Programs[15].Commands[3].CommandType := DUT_CommandType.MoveCommand;
PersistentVars.Programs[15].Commands[3].CommandString := 'DIR ABS 30.0 ACS LIT -19.65 30.42 -55.18 0.0 4.04 0.0 ';
PersistentVars.Programs[15].Commands[3].CommandComment := 'Taught position';
PersistentVars.Programs[15].Commands[6].CommandType := DUT_CommandType.VarSetCommand;
PersistentVars.Programs[15].Commands[6].CommandString := 'STO 46 E 0.0 E 0.0 E 300.0 E 0.0 E 0.0 E 0.0 ';
PersistentVars.Programs[15].Commands[6].CommandComment := 'offset the TCP Z';
PersistentVars.Programs[15].Commands[7].CommandType := DUT_CommandType.MoveCommand;
PersistentVars.Programs[15].Commands[7].CommandString := 'LIN ABS 20.0 TCS LIT 0.0 0.0 0.0 0.0 -30.0 0.0 ';
PersistentVars.Programs[15].Commands[7].CommandComment := 'rotate around TCP Y';
PersistentVars.Programs[15].Commands[8].CommandType := DUT_CommandType.MoveCommand;
PersistentVars.Programs[15].Commands[8].CommandString := 'LIN ABS 20.0 TCS LIT 0.0 0.0 0.0 90.0 60.0 -90.0 ';
PersistentVars.Programs[15].Commands[8].CommandComment := 'rotate around TCP X with z$' y z$'$'';
PersistentVars.Programs[15].Commands[10].CommandType := DUT_CommandType.MoveCommand;
PersistentVars.Programs[15].Commands[10].CommandString := 'DIR ABS 30.0 ACS LIT -19.65 30.42 -55.18 0.0 4.04 0.0 ';
PersistentVars.Programs[15].Commands[10].CommandComment := 'Taught position';
PersistentVars.Programs[15].Commands[12].CommandType := DUT_CommandType.VarSetCommand;
PersistentVars.Programs[15].Commands[12].CommandString := 'STO 43 E 100.0 E 1000.0 E 1000.0 E 1.0 E 1.0 E 1.0 ';
PersistentVars.Programs[15].Commands[12].CommandComment := 'set velocity, acceleration, and jerk';
                        
END_METHOD

METHOD PRIVATE _M_Controller : BOOL
VAR_INPUT
END_VAR
VAR_STAT
	_PowerRtrig: R_TRIG;
	_PowerFtrig: F_TRIG;
	_PowerTimerRtrig: R_TRIG;
	_PowerTimer: TON:=(PT:=T#1S);
	_PsButtonRtrig: R_TRIG;
	_PsButtonFtrig: F_TRIG;
	_PsButtonTimer: TON:=(PT:=T#2S);
	_PsButtonTimerRtrig: R_TRIG;
	_Reseting: BOOL;
END_VAR
                          
// dont get sleepy
Controller(sIpAddress:= '127.0.0.1', uPort:= 50013);

// put two fingers on the trackpad for 3 seconds to toggle power
_PowerTimer(IN:=Controller.P_State.Connected
				AND Controller.P_State.Buttons.Touch
				AND Controller.P_State.Trackpads.One.Active 
				AND Controller.P_State.Trackpads.Two.Active);
_PowerTimerRtrig(CLK:=_PowerTimer.Q);
IF _PowerTimerRtrig.Q THEN
	GVL.PowerOn := NOT GVL.PowerOn;
END_IF
_PowerRtrig(CLK:=GVL.Enable);
_PowerFtrig(CLK:=GVL.Enable);
IF _PowerRtrig.Q OR _PowerFtrig.Q THEN
	IF GVL.Enable THEN
		Controller.M_SetColor(255,0,0);
		Controller.M_SetBrightness(E_ControllerBrightness.High);
		Controller.M_SetMotorIntensity(E_ControllerMotor.Left, 100, 0.100);
	ELSE
		Controller.M_SetColor(0,255,0);
		Controller.M_SetBrightness(E_ControllerBrightness.Low);
		Controller.M_SetMotorIntensity(E_ControllerMotor.Right, 100, 0.100);
	END_IF
END_IF

// press PS button once to reset
_PsButtonRtrig(CLK:=Controller.P_State.Buttons.PS);
_PsButtonFtrig(CLK:=Controller.P_State.Buttons.PS);
IF _PsButtonRtrig.Q THEN
	_Reseting := TRUE;
END_IF
IF _PsButtonFtrig.Q THEN
	IF _Reseting THEN //  reset was not overridden by holding it down too long
		_Reseting := FALSE;
		GVL.Reset := TRUE;
	END_IF
END_IF

// hold down the PS button to home
_PsButtonTimer(IN:=Controller.P_State.Buttons.PS);
_PsButtonTimerRtrig(CLK:=_PsButtonTimer.Q);
IF _PsButtonTimerRtrig.Q THEN
	_Reseting := FALSE; // ps button was held down too long so we dont reset
	ProcessHome.M_StartHoming();
END_IF
                        
END_METHOD

METHOD PRIVATE _M_Tuning : BOOL
VAR_INPUT
END_VAR
VAR_STAT
	_MoveDelayTimer: ARRAY[0..5] OF TON;
	_TraceStartFtrig: ARRAY[0..5] OF F_TRIG;
	_MoveBusyFtrig: ARRAY[0..5] OF F_TRIG;
	_MoveBusyRtrig: ARRAY[0..5] OF R_TRIG;
	_MoveDelayTime: INT:=10; // ms
	_eDtState: ARRAY[0..5] OF INT; (* 0 idle, 1 wait cruise, 2 sampling, 3 done *)
	_bEstEnable: ARRAY[0..5] OF BOOL;
	_bDtFinish: ARRAY[0..5] OF BOOL;
	_aDtSample: ARRAY[0..5, 0..63] OF LREAL;
	_nSamples: ARRAY[0..5] OF INT;
	_fSetVel: LREAL;
	_fCruiseVel: LREAL;
	_fMedian: LREAL;
	_fSwap: LREAL;
	_fDtMin: LREAL := 0.1; (* SoftMotion rejects D = 0 *)
	_fDtMax: LREAL := 20.0; (* PosControl delay-buffer limit *)
	_fCruiseRatio: LREAL := 0.9;
	_nSampleMax: INT := 64;
	_bKpMode: ARRAY[0..5] OF BOOL;
	_bKpActive: ARRAY[0..5] OF BOOL;
	_bKpFinish: ARRAY[0..5] OF BOOL;
	_bKpApproached: ARRAY[0..5] OF BOOL;
	_fKpDist: ARRAY[0..5] OF LREAL;
	_fKpTarget: ARRAY[0..5] OF LREAL;
	_fKpActStart: ARRAY[0..5] OF LREAL;
	_fKpActMin: ARRAY[0..5] OF LREAL;
	_fKpActMax: ARRAY[0..5] OF LREAL;
	_fKpActLast: ARRAY[0..5] OF LREAL;
	_fKpPrevTgtErr: ARRAY[0..5] OF LREAL;
	_fKpPrevActDelta: ARRAY[0..5] OF LREAL;
	_fKpCruiseSum: ARRAY[0..5] OF LREAL;
	_nKpCruiseN: ARRAY[0..5] OF INT;
	_nKpSettle: ARRAY[0..5] OF INT;
	_bKpSettleInit: ARRAY[0..5] OF BOOL;
	_fKpSettleLeg: ARRAY[0..5] OF LREAL;
	_fSetPos: LREAL;
	_fActPos: LREAL;
	_fLag: LREAL;
	_fKpNow: LREAL;
	_fKpMin: LREAL := 0.0001;
	_fKpMax: LREAL := 2.0;
	_fKpRaise: LREAL := 1.5;
	_fKpLower: LREAL := 0.9;
	_fKpLagNoise: LREAL := 0.02;
	_fKpDeltaMin: LREAL := 0.003;
	_fKpBounceMin: LREAL := 0.08;
	_fKpApproachFrac: LREAL := 0.3;
	_fKpReachBand: LREAL := 0.15;
	_nKpSettleCycles: INT := 200;
	_i, _j, _k: INT;
END_VAR
                          // MainTask interval is the SoftMotion bus cycle that D is counted in.
// TaskInfo.dwInterval is microseconds (simulation writes 1000).
IF GVL.dwMainInterval > 0 THEN
	fCycleTimeMs := DWORD_TO_LREAL(GVL.dwMainInterval) / 1000.0;
ELSE
	fCycleTimeMs := 1.0;
END_IF

IF FirstScan THEN
	FOR _i:=0 TO 5 BY 1 DO
		sDeadTimeHelp[_i] := 'Kp=0 then START TUNE to estimate D. Kp>0 then START TUNE to score Kp.';
		sKpHelp[_i] := 'Set Kp above 0, WRITE PARAMETERS, then START TUNE to score overshoot and lag.';
		sKpVerdict[_i] := '';
	END_FOR
END_IF

// initial values
IF SetTuningMoveValues AND_THEN PersistentVars.Flags[GVL.INIT_DRV_IDX].Value THEN
	SetTuningMoveValues := FALSE;
	
	MoveRelative[0].Velocity := IoConfig_Globals.J1.fSWMaxVelocity;
	MoveRelative[0].Acceleration := IoConfig_Globals.J1.fSWMaxAcceleration;
	MoveRelative[0].Deceleration := IoConfig_Globals.J1.fSWMaxDeceleration;
	MoveRelative[0].Jerk := IoConfig_Globals.J1.fSWMaxJerk;
	MoveRelative[0].Distance := MoveDistance;
	
	MoveRelative[1].Velocity := IoConfig_Globals.J2.fSWMaxVelocity;
	MoveRelative[1].Acceleration := IoConfig_Globals.J2.fSWMaxAcceleration;
	MoveRelative[1].Deceleration := IoConfig_Globals.J2.fSWMaxDeceleration;
	MoveRelative[1].Jerk := IoConfig_Globals.J2.fSWMaxJerk;
	MoveRelative[1].Distance := MoveDistance;
	
	MoveRelative[2].Velocity := IoConfig_Globals.J3.fSWMaxVelocity;
	MoveRelative[2].Acceleration := IoConfig_Globals.J3.fSWMaxAcceleration;
	MoveRelative[2].Deceleration := IoConfig_Globals.J3.fSWMaxDeceleration;
	MoveRelative[2].Jerk := IoConfig_Globals.J3.fSWMaxJerk;
	MoveRelative[2].Distance := MoveDistance;
	
	MoveRelative[3].Velocity := IoConfig_Globals.J4.fSWMaxVelocity;
	MoveRelative[3].Acceleration := IoConfig_Globals.J4.fSWMaxAcceleration;
	MoveRelative[3].Deceleration := IoConfig_Globals.J4.fSWMaxDeceleration;
	MoveRelative[3].Jerk := IoConfig_Globals.J4.fSWMaxJerk;
	MoveRelative[3].Distance := MoveDistance;
	
	MoveRelative[4].Velocity := IoConfig_Globals.J5.fSWMaxVelocity;
	MoveRelative[4].Acceleration := IoConfig_Globals.J5.fSWMaxAcceleration;
	MoveRelative[4].Deceleration := IoConfig_Globals.J5.fSWMaxDeceleration;
	MoveRelative[4].Jerk := IoConfig_Globals.J5.fSWMaxJerk;
	MoveRelative[4].Distance := MoveDistance;
	
	MoveRelative[5].Velocity := IoConfig_Globals.J6.fSWMaxVelocity;
	MoveRelative[5].Acceleration := IoConfig_Globals.J6.fSWMaxAcceleration;
	MoveRelative[5].Deceleration := IoConfig_Globals.J6.fSWMaxDeceleration;
	MoveRelative[5].Jerk := IoConfig_Globals.J6.fSWMaxJerk;
	MoveRelative[5].Distance := MoveDistance;
END_IF

// trace activation
FOR _i:=0 TO 5 BY 1 DO
	
	IF TuneStart[_i] THEN
		TuneStart[_i] := FALSE;
		TraceStart[_i] := TRUE; // trace will handshake this bit low
		GroupHandler.M_EnableGroup();
		_bKpMode[_i] := PersistentVars.PositionControllers[_i].fKp > 0.0;
		bDeadTimeSuggested[_i] := FALSE;
		fMeasuredLagMs[_i] := 0.0;
		fEstimatedDeadTimeRaw[_i] := 0.0;
		fSuggestedDeadTime[_i] := 0.0;
		nDeadTimeSamples[_i] := 0;
		_eDtState[_i] := 0;
		_bEstEnable[_i] := FALSE;
		_bDtFinish[_i] := FALSE;
		_nSamples[_i] := 0;
		bKpSuggested[_i] := FALSE;
		fSuggestedKp[_i] := 0.0;
		fKpPeakLag[_i] := 0.0;
		fKpCruiseLag[_i] := 0.0;
		fKpFinalLag[_i] := 0.0;
		fKpOvershoot[_i] := 0.0;
		fKpUndershoot[_i] := 0.0;
		nKpReversals[_i] := 0;
		nKpVelReversals[_i] := 0;
		sKpVerdict[_i] := '';
		_bKpActive[_i] := FALSE;
		_bKpFinish[_i] := FALSE;
		_bKpApproached[_i] := FALSE;
		_nKpSettle[_i] := 0;
		_bKpSettleInit[_i] := FALSE;
		_fKpSettleLeg[_i] := 0.0;
		IF _bKpMode[_i] THEN
			sDeadTimeHelp[_i] := 'Kp tune: scoring this move. D is left unchanged.';
			sKpHelp[_i] := 'Scoring current Kp. Watch set vs actual; a suggestion appears when the move ends.';
		ELSE
			sDeadTimeHelp[_i] := 'SMC_EstimateDeadTime: waiting for constant velocity. Kp=0 gives the cleanest estimate.';
			sKpHelp[_i] := 'Kp is 0, so this pass estimates D only.';
		END_IF
	END_IF
	
	// copy a valid suggestion into the DeadTime spin; WRITE PARAMETERS still applies it
	IF UseSuggestedD[_i] THEN
		UseSuggestedD[_i] := FALSE;
		IF bDeadTimeSuggested[_i] THEN
			PersistentVars.PositionControllers[_i].fDeadTime := fSuggestedDeadTime[_i];
			sDeadTimeHelp[_i] := 'Copied suggested D into DeadTime. Press WRITE PARAMETERS to apply.';
		ELSE
			sDeadTimeHelp[_i] := 'No suggested D yet. Press START TUNE first.';
		END_IF
	END_IF
	
	IF UseSuggestedKp[_i] THEN
		UseSuggestedKp[_i] := FALSE;
		IF bKpSuggested[_i] THEN
			PersistentVars.PositionControllers[_i].fKp := fSuggestedKp[_i];
			sKpHelp[_i] := 'Copied suggested Kp. Press WRITE PARAMETERS to apply.';
		ELSE
			sKpHelp[_i] := 'No suggested Kp yet. Set Kp>0, WRITE PARAMETERS, then START TUNE.';
		END_IF
	END_IF
	
	IF RaiseKp[_i] THEN
		RaiseKp[_i] := FALSE;
		_fKpNow := PersistentVars.PositionControllers[_i].fKp;
		IF _fKpNow < _fKpMin THEN
			_fKpNow := _fKpMin;
		END_IF
		fSuggestedKp[_i] := _fKpNow * _fKpRaise;
		IF fSuggestedKp[_i] > _fKpMax THEN
			fSuggestedKp[_i] := _fKpMax;
		END_IF
		PersistentVars.PositionControllers[_i].fKp := fSuggestedKp[_i];
		bKpSuggested[_i] := TRUE;
		sKpVerdict[_i] := 'RAISED';
		sKpHelp[_i] := 'Raised Kp to ';
		sKpHelp[_i] := CONCAT(sKpHelp[_i], TO_STRING(fSuggestedKp[_i]));
		sKpHelp[_i] := CONCAT(sKpHelp[_i], '. WRITE PARAMETERS, START TUNE, watch the graph. When it fluctuates, press LOWER.');
	END_IF
	
	IF LowerKp[_i] THEN
		LowerKp[_i] := FALSE;
		_fKpNow := PersistentVars.PositionControllers[_i].fKp;
		fSuggestedKp[_i] := _fKpNow * _fKpLower;
		IF fSuggestedKp[_i] < _fKpMin THEN
			fSuggestedKp[_i] := _fKpMin;
		END_IF
		PersistentVars.PositionControllers[_i].fKp := fSuggestedKp[_i];
		bKpSuggested[_i] := TRUE;
		sKpVerdict[_i] := 'LOWERED';
		sKpHelp[_i] := 'Lowered Kp to ';
		sKpHelp[_i] := CONCAT(sKpHelp[_i], TO_STRING(fSuggestedKp[_i]));
		sKpHelp[_i] := CONCAT(sKpHelp[_i], '. WRITE PARAMETERS, then START TUNE. Official finish is ~10% below the first fluctuation.');
	END_IF
	
	// TraceStart will clear after handshake. this means the trace has started collecting samples
	// start the move delay timer to capture samples before the move
	_TraceStartFtrig[_i](CLK:=TraceStart[_i]);
	IF _TraceStartFtrig[_i].Q THEN
		_MoveDelayTimer[_i].IN:=TRUE;
	END_IF
	
	// once the move delay expires, start the move
	_MoveDelayTimer[_i](PT:=INT_TO_TIME(_MoveDelayTime));
	IF _MoveDelayTimer[_i].Q THEN
		_MoveDelayTimer[_i].IN:=FALSE;
		MoveRelative[_i].Execute := TRUE;
	END_IF
	
	_MoveBusyFtrig[_i](CLK:=MoveRelative[_i].Busy);
	IF _MoveBusyFtrig[_i].Q THEN
		MoveRelative[_i].Execute := FALSE;
		MoveRelative[_i].Distance := MoveRelative[_i].Distance * -1.0; // reverse direction
		_bEstEnable[_i] := FALSE;
		IF _bKpMode[_i] THEN
			_nKpSettle[_i] := _nKpSettleCycles;
			_bKpSettleInit[_i] := TRUE;
			sKpHelp[_i] := 'Move done, watching settle for a real bounce...';
		ELSIF _eDtState[_i] = 2 THEN
			_bDtFinish[_i] := TRUE;
		ELSIF _eDtState[_i] = 1 THEN
			_eDtState[_i] := 0;
			sDeadTimeHelp[_i] := 'Move ended before constant velocity. Increase MoveDistance or reduce acceleration.';
		END_IF
	END_IF

	CASE _i OF
		0:
			_fSetVel := IoConfig_Globals.J1.fSetVelocity;
			_fSetPos := IoConfig_Globals.J1.fSetPosition;
			_fActPos := IoConfig_Globals.J1.fActPosition;
		1:
			_fSetVel := IoConfig_Globals.J2.fSetVelocity;
			_fSetPos := IoConfig_Globals.J2.fSetPosition;
			_fActPos := IoConfig_Globals.J2.fActPosition;
		2:
			_fSetVel := IoConfig_Globals.J3.fSetVelocity;
			_fSetPos := IoConfig_Globals.J3.fSetPosition;
			_fActPos := IoConfig_Globals.J3.fActPosition;
		3:
			_fSetVel := IoConfig_Globals.J4.fSetVelocity;
			_fSetPos := IoConfig_Globals.J4.fSetPosition;
			_fActPos := IoConfig_Globals.J4.fActPosition;
		4:
			_fSetVel := IoConfig_Globals.J5.fSetVelocity;
			_fSetPos := IoConfig_Globals.J5.fSetPosition;
			_fActPos := IoConfig_Globals.J5.fActPosition;
		5:
			_fSetVel := IoConfig_Globals.J6.fSetVelocity;
			_fSetPos := IoConfig_Globals.J6.fSetPosition;
			_fActPos := IoConfig_Globals.J6.fActPosition;
	END_CASE
	
	_MoveBusyRtrig[_i](CLK:=MoveRelative[_i].Busy);
	IF _MoveBusyRtrig[_i].Q THEN
		IF _bKpMode[_i] THEN
			_bKpActive[_i] := TRUE;
			_bKpApproached[_i] := FALSE;
			_bKpFinish[_i] := FALSE;
			_nKpSettle[_i] := 0;
			_fKpDist[_i] := MoveRelative[_i].Distance;
			_fKpTarget[_i] := _fActPos + MoveRelative[_i].Distance;
			_fKpActStart[_i] := _fActPos;
			_fKpActMin[_i] := _fActPos;
			_fKpActMax[_i] := _fActPos;
			_fKpActLast[_i] := _fActPos;
			_fKpPrevTgtErr[_i] := 0.0;
			_fKpPrevActDelta[_i] := 0.0;
			_fKpCruiseSum[_i] := 0.0;
			_nKpCruiseN[_i] := 0;
			fKpPeakLag[_i] := 0.0;
			fKpCruiseLag[_i] := 0.0;
			fKpFinalLag[_i] := 0.0;
			fKpOvershoot[_i] := 0.0;
			fKpUndershoot[_i] := 0.0;
			nKpReversals[_i] := 0;
			nKpVelReversals[_i] := 0;
		ELSE
			_nSamples[_i] := 0;
			nDeadTimeSamples[_i] := 0;
			_bDtFinish[_i] := FALSE;
			_eDtState[_i] := 1;
		END_IF
	END_IF
	
	IF _bKpActive[_i] THEN
		_fLag := _fSetPos - _fActPos;
		IF ABS(_fLag) > fKpPeakLag[_i] THEN
			fKpPeakLag[_i] := ABS(_fLag);
		END_IF
		IF ABS(_fSetVel) >= (MoveRelative[_i].Velocity * _fCruiseRatio) THEN
			_fKpCruiseSum[_i] := _fKpCruiseSum[_i] + ABS(_fLag);
			_nKpCruiseN[_i] := _nKpCruiseN[_i] + 1;
		END_IF
		IF _fActPos < _fKpActMin[_i] THEN
			_fKpActMin[_i] := _fActPos;
		END_IF
		IF _fActPos > _fKpActMax[_i] THEN
			_fKpActMax[_i] := _fActPos;
		END_IF
		IF _bKpSettleInit[_i] THEN
			_bKpSettleInit[_i] := FALSE;
			_fKpActLast[_i] := _fActPos;
			_fKpSettleLeg[_i] := 0.0;
			nKpVelReversals[_i] := 0;
		ELSIF _nKpSettle[_i] > 0 THEN
			_fKpNow := _fActPos - _fKpActLast[_i];
			_fKpActLast[_i] := _fActPos;
			IF ABS(_fKpNow) > _fKpDeltaMin THEN
				IF (_fKpSettleLeg[_i] = 0.0) OR ((_fKpSettleLeg[_i] > 0.0) = (_fKpNow > 0.0)) THEN
					_fKpSettleLeg[_i] := _fKpSettleLeg[_i] + _fKpNow;
				ELSE
					IF ABS(_fKpSettleLeg[_i]) > _fKpBounceMin THEN
						nKpVelReversals[_i] := nKpVelReversals[_i] + 1;
					END_IF
					_fKpSettleLeg[_i] := _fKpNow;
				END_IF
			END_IF
		END_IF
		IF _nKpSettle[_i] > 0 THEN
			_nKpSettle[_i] := _nKpSettle[_i] - 1;
			IF _nKpSettle[_i] = 0 THEN
				_bKpFinish[_i] := TRUE;
			END_IF
		END_IF
	END_IF
	
	IF _bKpFinish[_i] THEN
		_bKpFinish[_i] := FALSE;
		_bKpActive[_i] := FALSE;
		_nKpSettle[_i] := 0;
		fKpFinalLag[_i] := ABS(_fKpTarget[_i] - _fActPos);
		IF _nKpCruiseN[_i] > 0 THEN
			fKpCruiseLag[_i] := _fKpCruiseSum[_i] / INT_TO_LREAL(_nKpCruiseN[_i]);
		ELSE
			fKpCruiseLag[_i] := fKpPeakLag[_i];
		END_IF
		IF _fKpDist[_i] >= 0.0 THEN
			fKpOvershoot[_i] := _fKpActMax[_i] - _fKpTarget[_i];
			fKpUndershoot[_i] := _fKpTarget[_i] - _fKpActMax[_i];
		ELSE
			fKpOvershoot[_i] := _fKpTarget[_i] - _fKpActMin[_i];
			fKpUndershoot[_i] := _fKpActMin[_i] - _fKpTarget[_i];
		END_IF
		IF fKpOvershoot[_i] < 0.0 THEN
			fKpOvershoot[_i] := 0.0;
		END_IF
		IF fKpUndershoot[_i] < 0.0 THEN
			fKpUndershoot[_i] := 0.0;
		END_IF
		_fKpNow := PersistentVars.PositionControllers[_i].fKp;
		IF nKpVelReversals[_i] >= 1 THEN
			sKpVerdict[_i] := 'TOO HOT';
			fSuggestedKp[_i] := _fKpNow * _fKpLower;
		ELSIF fKpUndershoot[_i] > _fKpReachBand THEN
			sKpVerdict[_i] := 'TOO SOFT';
			fSuggestedKp[_i] := _fKpNow * _fKpRaise;
		ELSE
			sKpVerdict[_i] := 'GOOD';
			fSuggestedKp[_i] := _fKpNow;
		END_IF
		IF fSuggestedKp[_i] < _fKpMin THEN
			fSuggestedKp[_i] := _fKpMin;
		ELSIF fSuggestedKp[_i] > _fKpMax THEN
			fSuggestedKp[_i] := _fKpMax;
		END_IF
		bKpSuggested[_i] := TRUE;
		sKpHelp[_i] := CONCAT(sKpVerdict[_i], '  und ');
		sKpHelp[_i] := CONCAT(sKpHelp[_i], TO_STRING(fKpUndershoot[_i]));
		sKpHelp[_i] := CONCAT(sKpHelp[_i], '  ov ');
		sKpHelp[_i] := CONCAT(sKpHelp[_i], TO_STRING(fKpOvershoot[_i]));
		sKpHelp[_i] := CONCAT(sKpHelp[_i], '  bounce ');
		sKpHelp[_i] := CONCAT(sKpHelp[_i], INT_TO_STRING(nKpVelReversals[_i]));
		sKpHelp[_i] := CONCAT(sKpHelp[_i], '  try Kp ');
		sKpHelp[_i] := CONCAT(sKpHelp[_i], TO_STRING(fSuggestedKp[_i]));
		sKpHelp[_i] := CONCAT(sKpHelp[_i], '. GOOD means this move did not bounce or miss. Use RAISE/LOWER and the graph.');
	END_IF
	
	_fCruiseVel := MoveRelative[_i].Velocity * _fCruiseRatio;
	IF (NOT _bKpMode[_i]) AND (_eDtState[_i] = 1) THEN
		IF ABS(_fSetVel) >= _fCruiseVel THEN
			_bEstEnable[_i] := TRUE;
			_eDtState[_i] := 2;
			sDeadTimeHelp[_i] := 'SMC_EstimateDeadTime: sampling at constant velocity...';
		END_IF
	END_IF
	
	IF _eDtState[_i] = 2 THEN
		IF _bEstEnable[_i] AND EstimateDeadTime[_i].Valid AND (_nSamples[_i] < _nSampleMax) THEN
			_aDtSample[_i, _nSamples[_i]] := ABS(EstimateDeadTime[_i].DeadTimeCycles);
			_nSamples[_i] := _nSamples[_i] + 1;
			nDeadTimeSamples[_i] := _nSamples[_i];
			IF _nSamples[_i] >= _nSampleMax THEN
				_bDtFinish[_i] := TRUE;
			END_IF
		END_IF
	END_IF
	
	IF _bDtFinish[_i] THEN
		_bDtFinish[_i] := FALSE;
		_bEstEnable[_i] := FALSE;
		_eDtState[_i] := 3;
		IF _nSamples[_i] < 1 THEN
			_eDtState[_i] := 0;
			sDeadTimeHelp[_i] := 'SMC_EstimateDeadTime never went Valid. Check enable and that the axis reached cruise.';
		ELSE
			// median of collected DeadTimeCycles
			FOR _j:=0 TO (_nSamples[_i] - 2) BY 1 DO
				FOR _k:=(_j + 1) TO (_nSamples[_i] - 1) BY 1 DO
					IF _aDtSample[_i, _k] < _aDtSample[_i, _j] THEN
						_fSwap := _aDtSample[_i, _j];
						_aDtSample[_i, _j] := _aDtSample[_i, _k];
						_aDtSample[_i, _k] := _fSwap;
					END_IF
				END_FOR
			END_FOR
			_fMedian := ABS(_aDtSample[_i, _nSamples[_i] / 2]);
			fEstimatedDeadTimeRaw[_i] := _fMedian;
			fMeasuredLagMs[_i] := _fMedian * fCycleTimeMs;
			IF _fMedian < _fDtMin THEN
				fSuggestedDeadTime[_i] := _fDtMin;
			ELSIF _fMedian > _fDtMax THEN
				fSuggestedDeadTime[_i] := _fDtMax;
			ELSE
				fSuggestedDeadTime[_i] := _fMedian;
			END_IF
			bDeadTimeSuggested[_i] := TRUE;
			sDeadTimeHelp[_i] := 'SMC_EstimateDeadTime median ';
			sDeadTimeHelp[_i] := CONCAT(sDeadTimeHelp[_i], TO_STRING(fEstimatedDeadTimeRaw[_i]));
			sDeadTimeHelp[_i] := CONCAT(sDeadTimeHelp[_i], ' cycles (');
			sDeadTimeHelp[_i] := CONCAT(sDeadTimeHelp[_i], TO_STRING(fMeasuredLagMs[_i]));
			sDeadTimeHelp[_i] := CONCAT(sDeadTimeHelp[_i], ' ms, n=');
			sDeadTimeHelp[_i] := CONCAT(sDeadTimeHelp[_i], INT_TO_STRING(_nSamples[_i]));
			IF fEstimatedDeadTimeRaw[_i] > _fDtMax THEN
				sDeadTimeHelp[_i] := CONCAT(sDeadTimeHelp[_i], '). Clamped to D 20 (PosControl max). WRITE PARAMETERS to apply.');
			ELSE
				sDeadTimeHelp[_i] := CONCAT(sDeadTimeHelp[_i], '). Suggested D ');
				sDeadTimeHelp[_i] := CONCAT(sDeadTimeHelp[_i], TO_STRING(fSuggestedDeadTime[_i]));
				sDeadTimeHelp[_i] := CONCAT(sDeadTimeHelp[_i], '. WRITE PARAMETERS to apply.');
			END_IF
		END_IF
	END_IF

END_FOR


// official SoftMotion estimator: enable only while at constant velocity
EstimateDeadTime[0](Axis:= IoConfig_Globals.J1, Enable:= _bEstEnable[0]);
EstimateDeadTime[1](Axis:= IoConfig_Globals.J2, Enable:= _bEstEnable[1]);
EstimateDeadTime[2](Axis:= IoConfig_Globals.J3, Enable:= _bEstEnable[2]);
EstimateDeadTime[3](Axis:= IoConfig_Globals.J4, Enable:= _bEstEnable[3]);
EstimateDeadTime[4](Axis:= IoConfig_Globals.J5, Enable:= _bEstEnable[4]);
EstimateDeadTime[5](Axis:= IoConfig_Globals.J6, Enable:= _bEstEnable[5]);

// move relative
MoveRelative[0](
	Axis:= IoConfig_Globals.J1, 
	Execute:= , 
	Distance:= , 
	Velocity:= , 
	Acceleration:= , 
	Deceleration:= , 
	Jerk:= , 
	BufferMode:= , 
	Done=> , 
	Busy=> , 
	Active=> , 
	CommandAborted=> , 
	Error=> , 
	ErrorID=> );
MoveRelative[1](
	Axis:= IoConfig_Globals.J2, 
	Execute:= , 
	Distance:= , 
	Velocity:= , 
	Acceleration:= , 
	Deceleration:= , 
	Jerk:= , 
	BufferMode:= , 
	Done=> , 
	Busy=> , 
	Active=> , 
	CommandAborted=> , 
	Error=> , 
	ErrorID=> );
MoveRelative[2](
	Axis:= IoConfig_Globals.J3, 
	Execute:= , 
	Distance:= , 
	Velocity:= , 
	Acceleration:= , 
	Deceleration:= , 
	Jerk:= , 
	BufferMode:= , 
	Done=> , 
	Busy=> , 
	Active=> , 
	CommandAborted=> , 
	Error=> , 
	ErrorID=> );
MoveRelative[3](
	Axis:= IoConfig_Globals.J4, 
	Execute:= , 
	Distance:= , 
	Velocity:= , 
	Acceleration:= , 
	Deceleration:= , 
	Jerk:= , 
	BufferMode:= , 
	Done=> , 
	Busy=> , 
	Active=> , 
	CommandAborted=> , 
	Error=> , 
	ErrorID=> );
MoveRelative[4](
	Axis:= IoConfig_Globals.J5, 
	Execute:= , 
	Distance:= , 
	Velocity:= , 
	Acceleration:= , 
	Deceleration:= , 
	Jerk:= , 
	BufferMode:= , 
	Done=> , 
	Busy=> , 
	Active=> , 
	CommandAborted=> , 
	Error=> , 
	ErrorID=> );
MoveRelative[5](
	Axis:= IoConfig_Globals.J6, 
	Execute:= , 
	Distance:= , 
	Velocity:= , 
	Acceleration:= , 
	Deceleration:= , 
	Jerk:= , 
	BufferMode:= , 
	Done=> , 
	Busy=> , 
	Active=> , 
	CommandAborted=> , 
	Error=> , 
	ErrorID=> );
                        
END_METHOD

METHOD PRIVATE _M_GroupHandler : BOOL
VAR_INPUT
END_VAR
                          
GroupHandler(
	AxisGroup:= ArfBotAxisGroup,
	Enable:= GVL.Enable,
	StoredPositions:= PersistentVars.StoredPositions,
	Busy=> , 
	Error=> , 
	ErrorID=> );
                        
END_METHOD
END_PROGRAM

PROGRAM _10_Robot
VAR	
	//
	AR4Inputs: ARRAY [0..31] OF BYTE;
	AR4Outputs: ARRAY [0..31] OF BYTE;
	
	//
	rx_heartbeat: BOOL;
	rx_en: BOOL;
	rx_j1_limit, rx_j2_limit, rx_j3_limit: BOOL;
	rx_j4_limit, rx_j5_limit, rx_j6_limit: BOOL;
	
	//
	InitializeDrives: BOOL;
	
	//
	FirstScan: BOOL:=TRUE;
	
END_VAR

                    //
IF FirstScan THEN
	M_Init(FALSE);
END_IF

_M_Init();
_M_HandleIO();

// do not put anything below this
FirstScan := FALSE;
                  

METHOD PRIVATE _M_HandleIO
VAR_INST
	//
	TxCrc, RxCrc: UINT;
	ChecksumMisCount: INT;
	
	//
	HeartbeatOn: TON;
	HeartbeatOff: TON;
	HeartbeatPt: TIME:=T#1000MS;
	
	//
	AR4OperationalFtrig: F_TRIG;
	
	//
	AllDrivesEnabled: BOOL;
	DriveEnable: ARRAY [0..5] OF BOOL;
	SetVelocity: ARRAY [0..5] OF INT;
	EncPosition: ARRAY [0..5] OF DINT;
	bufferIdx: INT;
	jointIdx: INT;
    
    //
    DeviceID: BYTE;
    RobotDeviceID: BYTE:=1;
	
END_VAR
                          //
HeartbeatOn(in:=NOT HeartbeatOff.Q,PT:=HeartbeatPt);
HeartbeatOff(in:=HeartbeatOn.Q,PT:=HeartbeatPt);

// if ethercat coms drop, clear the axes home status
{IF defined (IsSimulationMode)}
AR4OperationalFtrig(CLK:=TRUE);
{ELSE}
AR4OperationalFtrig(CLK:=AR4.wState = ETC_SLAVE_STATE.ETC_SLAVE_OPERATIONAL);
{END_IF}
IF AR4OperationalFtrig.Q THEN
	PersistentVars.Flags[GVL.HOME_COMPLETE].Value := FALSE;
	GVL.PowerOn := FALSE;
END_IF

// iSetVelocity is scaled counts, NOT °/s after the SoftMotion remap.
// deg/s = iSetVelocity * (MaxTU / MaxInt)
// Hz    = deg/s * StepsPerRev / 360

SetVelocity[0] := F_RoundToInt(
    (INT_TO_LREAL(IoConfig_Globals.J1.out.iSetVelocity) * GVL.c_PosCtrl_VelScale)
    * PersistentVars.PulsesPerRevolution[0] / 360.0);

SetVelocity[1] := F_RoundToInt(
    (INT_TO_LREAL(IoConfig_Globals.J2.out.iSetVelocity) * GVL.c_PosCtrl_VelScale)
    * PersistentVars.PulsesPerRevolution[1] / 360.0);

SetVelocity[2] := F_RoundToInt(
    (INT_TO_LREAL(IoConfig_Globals.J3.out.iSetVelocity) * GVL.c_PosCtrl_VelScale)
    * PersistentVars.PulsesPerRevolution[2] / 360.0);

SetVelocity[3] := F_RoundToInt(
    (INT_TO_LREAL(IoConfig_Globals.J4.out.iSetVelocity) * GVL.c_PosCtrl_VelScale)
    * PersistentVars.PulsesPerRevolution[3] / 360.0);

SetVelocity[4] := F_RoundToInt(
    (INT_TO_LREAL(IoConfig_Globals.J5.out.iSetVelocity) * GVL.c_PosCtrl_VelScale)
    * PersistentVars.PulsesPerRevolution[4] / 360.0);

SetVelocity[5] := F_RoundToInt(
    (INT_TO_LREAL(IoConfig_Globals.J6.out.iSetVelocity) * GVL.c_PosCtrl_VelScale)
    * PersistentVars.PulsesPerRevolution[5] / 360.0);

{region 'Output'}
// check that we are talking to the right device type
IF DeviceID = RobotDeviceID THEN// index 0 is for system outputs
    AR4Outputs[0].0:=HeartbeatOn.Q; // send a heartbeat to the drive
    AR4Outputs[0].1:=GVL.Enable; //
    // AR4Outputs[0].2:=; //
    // AR4Outputs[0].3:=; //
    // AR4Outputs[0].4:=; //
    // AR4Outputs[0].5:=; //
    // AR4Outputs[0].6:=; //
    // AR4Outputs[0].7:=; //
    
    // bytes 1 through 12 is for velocity to drive
    bufferIdx := 1;
    FOR jointIdx := 0 TO 5 BY 1 DO
        MEMUtils.MemCpy(pbyDest:=ADR(AR4Outputs[bufferIdx]), 
                        pbySrc:=ADR(SetVelocity[jointIdx]), 
                        dwSize:=SIZEOF(SetVelocity[jointIdx]));
        bufferIdx := bufferIdx + 2;
    END_FOR
    
    // bytes 13 through 24 are used for control from NC
    DriveEnable[0] := NOT (IoConfig_Globals.J1.nAxisState = SMC_AXIS_STATE.errorstop) AND NOT (IoConfig_Globals.J1.nAxisState = SMC_AXIS_STATE.power_off);
    DriveEnable[1] := NOT (IoConfig_Globals.J2.nAxisState = SMC_AXIS_STATE.errorstop) AND NOT (IoConfig_Globals.J2.nAxisState = SMC_AXIS_STATE.power_off);
    DriveEnable[2] := NOT (IoConfig_Globals.J3.nAxisState = SMC_AXIS_STATE.errorstop) AND NOT (IoConfig_Globals.J3.nAxisState = SMC_AXIS_STATE.power_off);
    DriveEnable[3] := NOT (IoConfig_Globals.J4.nAxisState = SMC_AXIS_STATE.errorstop) AND NOT (IoConfig_Globals.J4.nAxisState = SMC_AXIS_STATE.power_off);
    DriveEnable[4] := NOT (IoConfig_Globals.J5.nAxisState = SMC_AXIS_STATE.errorstop) AND NOT (IoConfig_Globals.J5.nAxisState = SMC_AXIS_STATE.power_off);
    DriveEnable[5] := NOT (IoConfig_Globals.J6.nAxisState = SMC_AXIS_STATE.errorstop) AND NOT (IoConfig_Globals.J6.nAxisState = SMC_AXIS_STATE.power_off);
    bufferIdx := 13;
    FOR jointIdx := 0 TO 5 BY 1 DO
        AR4Outputs[bufferIdx].3 := GVL.Enable AND DriveEnable[jointIdx];
        bufferIdx := bufferIdx + 1;
        // these are currently not used
        //AR4Outputs[bufferIdx].0 := Minus;
        //AR4Outputs[bufferIdx].1 := Plus;
        //AR4Outputs[bufferIdx].6 := Run;
        //AR4Outputs[bufferIdx].7 := Stop;
        bufferIdx := bufferIdx + 1;
    END_FOR
    
    // byte 25 is unused for now
    //AR4Outputs[25]:=;
    
    // byte 26 will be for gpio byte (bits 0 through 7)
    //AR4Outputs[26].0 := ;
    //AR4Outputs[26].1 := ;
    //AR4Outputs[26].2 := ;
    //AR4Outputs[26].3 := ;
    //AR4Outputs[26].4 := ;
    //AR4Outputs[26].5 := ;
    //AR4Outputs[26].6 := ;
    //AR4Outputs[26].7 := ;
    
    // bytes 27 through 28 are unused
    //AR4Outputs[27]:=;
    //AR4Outputs[28]:=;
    //AR4Outputs[29]:=;
    
    // byte 29 will be used to send the expected device id
    AR4Outputs[29] := RobotDeviceID;
    
END_IF

// bytes 30 and 31 will be used for crc
// calc crc here
TxCrc := F_Checksum(ADR(AR4Outputs), 30);
// append calc crc to tx buffer
MEMUtils.MemCpy(pbyDest:=ADR(AR4Outputs[30]), 
				pbySrc:=ADR(TxCrc), 
				dwSize:=2);
{endregion}
	
{region 'Input'}
// copy crc from rx buffer
MEMUtils.MemCpy(pbyDest:=ADR(RxCrc), 
				pbySrc:=ADR(AR4Inputs[30]), 
				dwSize:=2);

// compare calc crc with rx crc
{IF defined (IsSimulationMode)}
    PersistentVars.Flags[GVL.HOME_COMPLETE].Value := TRUE;
	rx_heartbeat := HeartbeatOn.Q;
	rx_en := GVL.Enable;
    EncPosition[0] := IoConfig_Globals.J1.diSetPosition;
    EncPosition[1] := IoConfig_Globals.J2.diSetPosition;
    EncPosition[2] := IoConfig_Globals.J3.diSetPosition;
    EncPosition[3] := IoConfig_Globals.J4.diSetPosition;
    EncPosition[4] := IoConfig_Globals.J5.diSetPosition;
    EncPosition[5] := IoConfig_Globals.J6.diSetPosition;
    rx_j1_limit :=
	rx_j2_limit :=
	rx_j3_limit :=
	rx_j4_limit :=
	rx_j5_limit :=
	rx_j6_limit :=
    IoConfig_Globals.J1.in.bDriveStartRealState :=
	IoConfig_Globals.J1.in.bRegulatorRealState :=
	IoConfig_Globals.J2.in.bDriveStartRealState :=
	IoConfig_Globals.J2.in.bRegulatorRealState :=
	IoConfig_Globals.J3.in.bDriveStartRealState :=
	IoConfig_Globals.J3.in.bRegulatorRealState :=
	IoConfig_Globals.J4.in.bDriveStartRealState :=
	IoConfig_Globals.J4.in.bRegulatorRealState :=
	IoConfig_Globals.J5.in.bDriveStartRealState :=
	IoConfig_Globals.J5.in.bRegulatorRealState :=
	IoConfig_Globals.J6.in.bDriveStartRealState :=
	IoConfig_Globals.J6.in.bRegulatorRealState :=
    AllDrivesEnabled := GVL.Enable;
    DeviceID := RobotDeviceID;
{ELSE}
IF RxCrc = F_Checksum(ADR(AR4Inputs), 30) THEN
	// byte 0 is for system inputs
	rx_heartbeat	:= AR4Inputs[0].0; // receive the heartbeat back
	rx_en 			:= AR4Inputs[0].1; // receive the enable back
	//rx_	 			:= AR4Inputs[0].2;
	//rx_ 				:= AR4Inputs[0].3;
	//rx_ 				:= AR4Inputs[0].4;
	//rx_ 				:= AR4Inputs[0].5;
	//rx_ 				:= AR4Inputs[0].6;
	//rx_ 				:= AR4Inputs[0].7;
	
	// bytes 1 through 24 is for encoder data from drive
	bufferIdx := 1;
	FOR jointIdx := 0 TO 5 BY 1 DO
		MEMUtils.MemCpy(pbyDest:=ADR(EncPosition[jointIdx]), 
						pbySrc:=ADR(AR4Inputs[bufferIdx]), 
						dwSize:=SIZEOF(EncPosition[jointIdx]));
		bufferIdx := bufferIdx + 4;
	END_FOR
	
	// byte 25 will be for limit switch inputs
	rx_j1_limit := AR4Inputs[25].0;
	rx_j2_limit := AR4Inputs[25].1;
	rx_j3_limit := AR4Inputs[25].2;
	rx_j4_limit := AR4Inputs[25].3;
	rx_j5_limit := AR4Inputs[25].4;
	rx_j6_limit := AR4Inputs[25].5;
	//rx_ := AR4Inputs[25].6;
	//rx_ := AR4Inputs[25].7;
	
	// byte 26 will be for gpio byte (bits 0 through 7)
	// := AR4Inputs[26].0;
	// := AR4Inputs[26].1;
	// := AR4Inputs[26].2;
	// := AR4Inputs[26].3;
	// := AR4Inputs[26].4;
	// := AR4Inputs[26].5;
	// := AR4Inputs[26].6;
	// := AR4Inputs[26].7;
	
	// byte 27 will be used to indicate drive is enabled
	IoConfig_Globals.J1.in.bDriveStartRealState := AR4Inputs[27].0;
	IoConfig_Globals.J1.in.bRegulatorRealState := AR4Inputs[27].0;
	IoConfig_Globals.J2.in.bDriveStartRealState := AR4Inputs[27].1;
	IoConfig_Globals.J2.in.bRegulatorRealState := AR4Inputs[27].1;
	IoConfig_Globals.J3.in.bDriveStartRealState := AR4Inputs[27].2;
	IoConfig_Globals.J3.in.bRegulatorRealState := AR4Inputs[27].2;
	IoConfig_Globals.J4.in.bDriveStartRealState := AR4Inputs[27].3;
	IoConfig_Globals.J4.in.bRegulatorRealState := AR4Inputs[27].3;
	IoConfig_Globals.J5.in.bDriveStartRealState := AR4Inputs[27].4;
	IoConfig_Globals.J5.in.bRegulatorRealState := AR4Inputs[27].4;
	IoConfig_Globals.J6.in.bDriveStartRealState := AR4Inputs[27].5;
	IoConfig_Globals.J6.in.bRegulatorRealState := AR4Inputs[27].5;
	// all drives are enabled
	AllDrivesEnabled := AR4Inputs[27].0 AND AR4Inputs[27].1 AND AR4Inputs[27].2
						AND AR4Inputs[27].3 AND AR4Inputs[27].4 AND AR4Inputs[27].5;
	
	// byte 28 is unused
	//
    
    // byte 29 will be used to identify the device
	DeviceID := AR4Inputs[29];
	
	// Rx buffer index 30 and 31 will be for crc
ELSE
	// increment crc mismatch counter
	ChecksumMisCount := ChecksumMisCount + 1;
END_IF
{END_IF}
{endregion}

// https://docs.google.com/spreadsheets/d/1S5TOxwbAx8pTMUdoWMnyC9WPfphhtUME/edit#gid=595805457
IoConfig_Globals.J1.in.dwActPosition := DINT_TO_DWORD(EncPosition[0]);
IoConfig_Globals.J2.in.dwActPosition := DINT_TO_DWORD(EncPosition[1]);
IoConfig_Globals.J3.in.dwActPosition := DINT_TO_DWORD(EncPosition[2]);
IoConfig_Globals.J4.in.dwActPosition := DINT_TO_DWORD(EncPosition[3]);
IoConfig_Globals.J5.in.dwActPosition := DINT_TO_DWORD(EncPosition[4]);
IoConfig_Globals.J6.in.dwActPosition := DINT_TO_DWORD(EncPosition[5]);

//
IF FirstScan THEN
	IoConfig_Globals.J1.bHWLimitEnable := TRUE;
	IoConfig_Globals.J2.bHWLimitEnable := TRUE;
	IoConfig_Globals.J3.bHWLimitEnable := TRUE;
	IoConfig_Globals.J4.bHWLimitEnable := TRUE;
	IoConfig_Globals.J5.bHWLimitEnable := TRUE;
	IoConfig_Globals.J6.bHWLimitEnable := TRUE;
END_IF

//
IoConfig_Globals.J1.in.bLimitNeg := TRUE;
IoConfig_Globals.J2.in.bLimitNeg := TRUE;
IoConfig_Globals.J3.in.bLimitNeg := rx_j3_limit;
IoConfig_Globals.J4.in.bLimitNeg := rx_j4_limit;
IoConfig_Globals.J5.in.bLimitNeg := rx_j5_limit;
IoConfig_Globals.J6.in.bLimitNeg := TRUE;

IoConfig_Globals.J1.in.bLimitPos := rx_j1_limit;
IoConfig_Globals.J2.in.bLimitPos := rx_j2_limit;
IoConfig_Globals.J3.in.bLimitPos := TRUE;
IoConfig_Globals.J4.in.bLimitPos := TRUE;
IoConfig_Globals.J5.in.bLimitPos := TRUE;
//IoConfig_Globals.J6.in.bLimitPos := rx_j6_limit;
// J6 home flag is not a travel stop — 360 deg tool-Z / cone orbits will cross it.
// Homing still uses rx_j6_limit as SMC_Homing.bReferenceSwitch (NOT J6_Limit).
IoConfig_Globals.J6.in.bLimitPos := TRUE;
                        
END_METHOD

METHOD PUBLIC M_Init : BOOL
VAR_INPUT
	DefaultParameters: BOOL;
END_VAR
                          IF DefaultParameters THEN
	PersistentVars.Flags[GVL.INIT_DRV_IDX].Value := FALSE;
END_IF
InitializeDrives := TRUE;
                        
END_METHOD

METHOD PRIVATE _M_Init
VAR_INPUT
END_VAR
VAR_STAT
	_Step: INT;
	_Done: BOOL;
	_Success: BOOL;
	_SMC_SetPosControlParams: ARRAY[0..5] OF SMC_SetPosControlParams;
	_i, _j, _k: INT;
END_VAR
                          
CASE _Step OF
	0:
		IF InitializeDrives THEN
			InitializeDrives := FALSE;
			//
			FOR _i:=GVL.POSCONT_ARR_BEG TO GVL.POSCONT_ARR_END BY 1 DO
				_SMC_SetPosControlParams[_i].bExecute := FALSE;
			END_FOR
			//
			IF NOT PersistentVars.Flags[GVL.INIT_DRV_IDX].Value THEN
				FOR _i:=GVL.POSCONT_ARR_BEG TO GVL.POSCONT_ARR_END BY 1 DO
					PersistentVars.PositionControllers[_i].fKp := 0.1;
					PersistentVars.PositionControllers[_i].fPartVelPilotControl := 1.0; // 0-1
					PersistentVars.PositionControllers[_i].fDeadTime := 2.0;
					PersistentVars.PositionControllers[_i].fMaxPositionDiff := 0.0;
					PersistentVars.PositionControllers[_i].fSWMaxVelocity := 30.0;
					PersistentVars.PositionControllers[_i].fSWMaxAcceleration := 1000.0;
					PersistentVars.PositionControllers[_i].fSWMaxDeceleration := 1000.0;
					PersistentVars.PositionControllers[_i].fSWMaxJerk := 10000.0;
				END_FOR
			END_IF
			// next, please
			_Step := _Step + 1;
		END_IF
		
	1: 
		//
		FOR _i:=GVL.POSCONT_ARR_BEG TO GVL.POSCONT_ARR_END BY 1 DO
			_SMC_SetPosControlParams[_i].bExecute := TRUE;
		END_FOR
		// next, please
		_Step := _Step + 1;
		
	2:
		//
		_Done := TRUE;
		_Success := TRUE;
		FOR _i:=GVL.POSCONT_ARR_BEG TO GVL.POSCONT_ARR_END BY 1 DO
			IF _SMC_SetPosControlParams[_i].bError THEN
				_Success := FALSE;
				EXIT;
			END_IF
			IF NOT _SMC_SetPosControlParams[_i].bDone THEN
				_Success := FALSE;
				_Done := FALSE;
				EXIT;
			END_IF
		END_FOR
		IF _Done THEN
			// next, please
			_Step := _Step + 1;
		END_IF
		
	3:
		//
		FOR _i:=GVL.POSCONT_ARR_BEG TO GVL.POSCONT_ARR_END BY 1 DO
			_SMC_SetPosControlParams[_i].bExecute := FALSE;
		END_FOR
		//
		IF _Success THEN
			PersistentVars.Flags[GVL.INIT_DRV_IDX].Value := TRUE;
		END_IF
		// next, please
		_Step := 0;
		
END_CASE

//
_SMC_SetPosControlParams[0](
	Axis:= IoConfig_Globals.J1, 
	bExecute:= , 
	fKp:= PersistentVars.PositionControllers[0].fKp, 
	fPartVelPilotControl:= PersistentVars.PositionControllers[0].fPartVelPilotControl, 
	fDeadTime:= PersistentVars.PositionControllers[0].fDeadTime, 
	fMaxPositionDiff:=PersistentVars.PositionControllers[0].fMaxPositionDiff, 
	bDone=> , 
	bError=> , 
	ErrorID=> );
IF _SMC_SetPosControlParams[0].bDone AND NOT _SMC_SetPosControlParams[0].bError THEN
	IoConfig_Globals.J1.fSWMaxVelocity 			:= PersistentVars.PositionControllers[0].fSWMaxVelocity; // 30
	IoConfig_Globals.J1.fSWMaxAcceleration 		:= PersistentVars.PositionControllers[0].fSWMaxAcceleration; // 1000
	IoConfig_Globals.J1.fSWMaxDeceleration 		:= PersistentVars.PositionControllers[0].fSWMaxDeceleration; // 1000
	IoConfig_Globals.J1.fSWMaxJerk 				:= PersistentVars.PositionControllers[0].fSWMaxJerk; // 10000
END_IF

//
_SMC_SetPosControlParams[1](
	Axis:= IoConfig_Globals.J2, 
	bExecute:= , 
	fKp:= PersistentVars.PositionControllers[1].fKp, 
	fPartVelPilotControl:= PersistentVars.PositionControllers[1].fPartVelPilotControl, 
	fDeadTime:= PersistentVars.PositionControllers[1].fDeadTime, 
	fMaxPositionDiff:=PersistentVars.PositionControllers[1].fMaxPositionDiff, 
	bDone=> , 
	bError=> , 
	ErrorID=> );
IF _SMC_SetPosControlParams[1].bDone AND NOT _SMC_SetPosControlParams[1].bError THEN
	IoConfig_Globals.J2.fSWMaxVelocity 			:= PersistentVars.PositionControllers[1].fSWMaxVelocity;
	IoConfig_Globals.J2.fSWMaxAcceleration 		:= PersistentVars.PositionControllers[1].fSWMaxAcceleration;
	IoConfig_Globals.J2.fSWMaxDeceleration 		:= PersistentVars.PositionControllers[1].fSWMaxDeceleration;
	IoConfig_Globals.J2.fSWMaxJerk 				:= PersistentVars.PositionControllers[1].fSWMaxJerk;
END_IF

//
_SMC_SetPosControlParams[2](
	Axis:= IoConfig_Globals.J3, 
	bExecute:= , 
	fKp:= PersistentVars.PositionControllers[2].fKp, 
	fPartVelPilotControl:= PersistentVars.PositionControllers[2].fPartVelPilotControl, 
	fDeadTime:= PersistentVars.PositionControllers[2].fDeadTime, 
	fMaxPositionDiff:=PersistentVars.PositionControllers[2].fMaxPositionDiff, 
	bDone=> , 
	bError=> , 
	ErrorID=> );
IF _SMC_SetPosControlParams[2].bDone AND NOT _SMC_SetPosControlParams[2].bError THEN
	IoConfig_Globals.J3.fSWMaxVelocity 			:= PersistentVars.PositionControllers[2].fSWMaxVelocity;
	IoConfig_Globals.J3.fSWMaxAcceleration 		:= PersistentVars.PositionControllers[2].fSWMaxAcceleration;
	IoConfig_Globals.J3.fSWMaxDeceleration 		:= PersistentVars.PositionControllers[2].fSWMaxDeceleration;
	IoConfig_Globals.J3.fSWMaxJerk 				:= PersistentVars.PositionControllers[2].fSWMaxJerk;
END_IF

//
_SMC_SetPosControlParams[3](
	Axis:= IoConfig_Globals.J4, 
	bExecute:= , 
	fKp:= PersistentVars.PositionControllers[3].fKp, 
	fPartVelPilotControl:= PersistentVars.PositionControllers[3].fPartVelPilotControl, 
	fDeadTime:= PersistentVars.PositionControllers[3].fDeadTime, 
	fMaxPositionDiff:=PersistentVars.PositionControllers[3].fMaxPositionDiff, 
	bDone=> , 
	bError=> , 
	ErrorID=> );
IF _SMC_SetPosControlParams[3].bDone AND NOT _SMC_SetPosControlParams[3].bError THEN
	IoConfig_Globals.J4.fSWMaxVelocity 			:= PersistentVars.PositionControllers[3].fSWMaxVelocity;
	IoConfig_Globals.J4.fSWMaxAcceleration 		:= PersistentVars.PositionControllers[3].fSWMaxAcceleration;
	IoConfig_Globals.J4.fSWMaxDeceleration 		:= PersistentVars.PositionControllers[3].fSWMaxDeceleration;
	IoConfig_Globals.J4.fSWMaxJerk 				:= PersistentVars.PositionControllers[3].fSWMaxJerk;
END_IF

//
_SMC_SetPosControlParams[4](
	Axis:= IoConfig_Globals.J5, 
	bExecute:= , 
	fKp:= PersistentVars.PositionControllers[4].fKp, 
	fPartVelPilotControl:= PersistentVars.PositionControllers[4].fPartVelPilotControl, 
	fDeadTime:= PersistentVars.PositionControllers[4].fDeadTime, 
	fMaxPositionDiff:=PersistentVars.PositionControllers[4].fMaxPositionDiff, 
	bDone=> , 
	bError=> , 
	ErrorID=> );
IF _SMC_SetPosControlParams[4].bDone AND NOT _SMC_SetPosControlParams[4].bError THEN
	IoConfig_Globals.J5.fSWMaxVelocity 			:= PersistentVars.PositionControllers[4].fSWMaxVelocity;
	IoConfig_Globals.J5.fSWMaxAcceleration 		:= PersistentVars.PositionControllers[4].fSWMaxAcceleration;
	IoConfig_Globals.J5.fSWMaxDeceleration 		:= PersistentVars.PositionControllers[4].fSWMaxDeceleration;
	IoConfig_Globals.J5.fSWMaxJerk 				:= PersistentVars.PositionControllers[4].fSWMaxJerk;
END_IF

//
_SMC_SetPosControlParams[5](
	Axis:= IoConfig_Globals.J6, 
	bExecute:= , 
	fKp:= PersistentVars.PositionControllers[5].fKp, 
	fPartVelPilotControl:= PersistentVars.PositionControllers[5].fPartVelPilotControl, 
	fDeadTime:= PersistentVars.PositionControllers[5].fDeadTime, 
	fMaxPositionDiff:=PersistentVars.PositionControllers[5].fMaxPositionDiff, 
	bDone=> , 
	bError=> , 
	ErrorID=> );
IF _SMC_SetPosControlParams[5].bDone AND NOT _SMC_SetPosControlParams[5].bError THEN
	IoConfig_Globals.J6.fSWMaxVelocity 			:= PersistentVars.PositionControllers[5].fSWMaxVelocity;
	IoConfig_Globals.J6.fSWMaxAcceleration 		:= PersistentVars.PositionControllers[5].fSWMaxAcceleration;
	IoConfig_Globals.J6.fSWMaxDeceleration 		:= PersistentVars.PositionControllers[5].fSWMaxDeceleration;
	IoConfig_Globals.J6.fSWMaxJerk 				:= PersistentVars.PositionControllers[5].fSWMaxJerk;
END_IF
                        
END_METHOD
END_PROGRAM

FUNCTION_BLOCK FB_JogProcessor
VAR_IN_OUT
	AxisGroup: AXIS_GROUP_REF_SM3;
	GroupHandler: FB_GroupHandler;
	Controller: FB_Controller;
END_VAR
VAR_INPUT
	Enable: BOOL;
	Reset: BOOL;
	StoredPositions: REFERENCE TO ARRAY[GVL.POS_ARR_BEG..GVL.POS_ARR_END] OF DUT_StoredPosition;
	VisionRegisters: REFERENCE TO ARRAY[GVL.VIS_ARR_BEG..GVL.VIS_ARR_END] OF DUT_VisionRegister;
	Flags: REFERENCE TO ARRAY[GVL.FLG_ARR_BEG..GVL.FLG_ARR_END] OF DUT_Flags;
END_VAR
VAR_OUTPUT
	ABC_as_ACS: BOOL;
	CoordSystem: SMC_COORD_SYSTEM;
	Position: SMC_POS_REF;
	Enabled: BOOL;
	Done: BOOL;
	Busy: BOOL;
	Error: BOOL;
	ErrorID: SMC_ERROR;
END_VAR
VAR
	_ExecuteRtrig: R_TRIG;
	_ExecuteFtrig: F_TRIG;
	_ResetRtrig: R_TRIG;
	_ErrorRtrig: R_TRIG;
	_EnableFtrig: F_TRIG;
	
	_SequenceMain: INT;
	_SequenceSetCoordTrans: INT;
	
	_SMC_GroupJog2: SMC_GroupJog2;
	
	_ControllerCenter: USINT:=128;
	_ControllerDeadZone: USINT:=40;
	
	_OffsetExist: ARRAY[0..GVL.MCS_POS_IDX-GVL.TCP_POS_IDX] OF BOOL;
	
	_MoveToPose: ARRAY[0..GVL.POSE_5_IDX-GVL.POSE_1_IDX] OF BOOL;
	_MoveCommandProcessor: FB_MoveCmdProcessor;
	
	_i, _j, _k: INT;
	_FirstScan: BOOL:=TRUE;
	
END_VAR

VAR CONSTANT
	STEP_DONE: 				INT := 1000;
	STEP_IDLE: 				INT := 0000;
	STEP_GROUP_ENABLE: 		INT := 0030;
	STEP_WAIT_ENABLE: 		INT := 0035;
	STEP_SET_KINEMATICS: 	INT := 0060;
	STEP_WAIT_KINEMATICS: 	INT := 0070;
	STEP_JOG:				INT := 0080;
	STEP_WAIT_JOG:			INT := 0090;
	STEP_GROUP_DISABLE: 	INT := 0100;
	STEP_WAIT_DISABLE: 		INT := 0110;
END_VAR

                    _ExecuteRtrig(CLK:=_SMC_GroupJog2.Enable);
_ExecuteFtrig(CLK:=_SMC_GroupJog2.Enable);
_ResetRtrig(CLK:=Reset);

IF _FirstScan THEN
	_SMC_GroupJog2.Velocity := 50.0;
	_SMC_GroupJog2.Acceleration := 300.0;
	_SMC_GroupJog2.Deceleration := 300.0;
	_SMC_GroupJog2.Jerk := 1000.0;
	_SMC_GroupJog2.MaxAngularDistance := 90.0;
	_SMC_GroupJog2.MaxLinearDistance := 200.0;
	_SMC_GroupJog2.AccFactor := 1.0;
	_SMC_GroupJog2.VelFactor := 0.1;
	_SMC_GroupJog2.JerkFactor := 1.0;
	_SMC_GroupJog2.TorqueFactor := 1.0;
	_SMC_GroupJog2.CoordSystem := SMC_COORD_SYSTEM.TCS;
	
END_IF

//
_M_HandleController(Controller:=Controller);
_M_HandlePose(AxisGroup:=AxisGroup, GroupHandler:=GroupHandler);

//
_EnableFtrig(CLK:=Enable);
IF _EnableFtrig.Q THEN
	_SMC_GroupJog2.Enable := FALSE;
END_IF

//
CASE _SequenceMain OF
	STEP_DONE: // done
		Busy := FALSE;
		Done := TRUE;
		_SequenceMain := STEP_IDLE;
		_MoveCommandProcessor.M_Home();
		
	STEP_IDLE: // IDLE
		IF _ExecuteRtrig.Q AND Enable THEN
			Busy := TRUE;
			Done := FALSE;
			_M_CheckOffsets();
			_SequenceMain := STEP_GROUP_ENABLE;
		END_IF
		
	STEP_GROUP_ENABLE:
		IF GroupHandler.M_EnableGroup() THEN
			_SequenceMain := STEP_WAIT_ENABLE;
		ELSE
			_SequenceMain := STEP_DONE;
			Error := TRUE;
			ErrorID := GroupHandler.ErrorID;
		END_IF
		
	STEP_WAIT_ENABLE:
		// TODO add timeout timer here
		IF GroupHandler.P_GroupEnabled THEN
			_SequenceMain := STEP_SET_KINEMATICS;
		END_IF;
		
	STEP_SET_KINEMATICS: // set kinematics
        // orientation convention is always ZYZ for softmotion
        GVL.OriConvention := SMC_ORI_CONVENTION.ZYZ;
        //
		IF GroupHandler.M_SetKinematics(_SMC_GroupJog2.CoordSystem) THEN
			_SequenceMain := STEP_WAIT_KINEMATICS;
		ELSE
			_SequenceMain := STEP_DONE;
			Error := TRUE;
			ErrorID := GroupHandler.ErrorID;
		END_IF
		
	STEP_WAIT_KINEMATICS:
		// TODO add timeout timer here
		IF GroupHandler.P_KinematicsSet THEN
			_SequenceMain := STEP_WAIT_JOG;
		END_IF
		
	STEP_WAIT_JOG: //
		IF _SMC_GroupJog2.Error THEN
			Error := TRUE;
			ErrorID := _SMC_GroupJog2.ErrorID;
		END_IF
		IF _ExecuteFtrig.Q THEN
			//_SequenceMain := STEP_GROUP_DISABLE;
			_SequenceMain := STEP_DONE;
		END_IF
		
	// TODO: do we need to disable the group at this point? lets leave this here for now but skip it.	
	STEP_GROUP_DISABLE:
		IF GroupHandler.M_DisableGroup() THEN
			_SequenceMain := STEP_WAIT_DISABLE;
		ELSE
			_SequenceMain := STEP_DONE;
			Error := TRUE;
			ErrorID := GroupHandler.ErrorID;
		END_IF
		
	STEP_WAIT_DISABLE:
		// TODO add timeouttimer here
		IF NOT GroupHandler.P_GroupEnabled THEN
			_SequenceMain := STEP_DONE;
		END_IF
	
END_CASE

//
IF _ResetRtrig.Q AND Error THEN
	Error := FALSE;
	ErrorID := SMC_NO_ERROR;
	_SequenceMain := STEP_DONE;
	GroupHandler.M_ResetGroup();
	_MoveCommandProcessor.M_Home();
END_IF

_SMC_GroupJog2(
	AxisGroup:= AxisGroup, 
	Enable:= , 
	Forward:= , 
	Backward:= , 
	MaxLinearDistance:= , 
	MaxAngularDistance:= , 
	Velocity:= , 
	Acceleration:= , 
	Deceleration:= , 
	Jerk:= , 
	VelFactor:= , 
	AccFactor:= , 
	JerkFactor:= , 
	TorqueFactor:= , 
	CoordSystem:= , 
	ABC_as_ACS:= , 
	Active=> , 
	Busy=> , 
	Error=> , 
	ErrorID=> , 
	CurrentPosition=> Position);

//
CoordSystem := _SMC_GroupJog2.CoordSystem;
ABC_as_ACS := _SMC_GroupJog2.ABC_as_ACS;
Enabled := _SMC_GroupJog2.Enable;

//
_ErrorRtrig(CLK:=GroupHandler.Error
				OR _SMC_GroupJog2.Error
				OR _MoveCommandProcessor.Error);			
IF _ErrorRtrig.Q THEN
	// TODO need to rework how error messages are handled (globally)
	// if the move command processor has an error, we dont know what it is.
	Error := TRUE;
END_IF

// do not put anything after this
_FirstScan := FALSE;
                  

METHOD PRIVATE _M_HandleController : BOOL
VAR_IN_OUT
	Controller: FB_Controller;
END_VAR
VAR_INPUT
END_VAR
VAR_STAT
	OptionsTimer: TON:=(PT:=T#1S);
	OptionsRtrig: R_TRIG;
	ShareTimer: TON:=(PT:=T#1S);
	ShareRtrig: R_TRIG;
	OptionsShareRtrig: R_TRIG;
	JogEnabledRtrig: R_TRIG;
	JogEnabledFtrig: F_TRIG;
	SquareButtonRtrig: R_TRIG;
	TriangleButtonRtrig: R_TRIG;
	CircleButtonRtrig: R_TRIG;
	CrossButtonRtrig: R_TRIG;
	R2_Last: USINT;
	JoyStickLeftXLast: USINT;
	JoyStickLeftYLast: USINT;
	JoyStickRightXLast: USINT;
	JoyStickRightYLast: USINT;
	FactorMin: LREAL:=0.01;
END_VAR
                          //
OptionsTimer(IN:=Controller.P_State.Buttons.Options);
OptionsRtrig(CLK:=Controller.P_State.Buttons.Options);
//
ShareTimer(IN:=Controller.P_State.Buttons.Share);
ShareRtrig(CLK:=Controller.P_State.Buttons.Share);
//
OptionsShareRtrig(CLK:=OptionsTimer.Q AND_THEN ShareTimer.Q);
JogEnabledRtrig(CLK:=_SMC_GroupJog2.Enable);
JogEnabledFtrig(CLK:=_SMC_GroupJog2.Enable);


IF Enable AND_THEN Controller.P_State.Connected THEN
	
	// toggle jog enable
	IF OptionsShareRtrig.Q THEN
		_SMC_GroupJog2.Enable := NOT _SMC_GroupJog2.Enable;
	END_IF
	IF JogEnabledRtrig.Q OR JogEnabledFtrig.Q THEN
		IF _SMC_GroupJog2.Enable THEN
			_SMC_GroupJog2.CoordSystem := SMC_COORD_SYSTEM.TCS;
			Controller.M_SetTriggerMode(E_ControllerTrigger.Right, E_ControllerTriggerMode.Rigid);
			Controller.M_SetTriggerForce(E_ControllerTrigger.Right, E_ControllerTriggerForceParameter.One, 0);
			Controller.M_SetPlayerID(E_ControllerPlayerID.PlayerALL);
			Controller.M_SetMicrophoneState(TRUE);
		ELSE
			Controller.M_SetTriggerMode(E_ControllerTrigger.Right, E_ControllerTriggerMode.Off);
			Controller.M_SetMicrophoneState(FALSE);
		END_IF
	END_IF
	
